Omron CX-Programmer project 新工程 (CX-Programmer 9.42)

# PLC HJ正压氦检: CJ2M CPU34
I/O table (CPU CJ2M-CPU34): rack 0 slot 0 CJ1W-NC413; rack 0 slot 1 CJ1W-SCU21-V1; rack 0 slot 2 CJ1W-AD081-V1; rack 0 slot 3 CJ1W-ID261; rack 0 slot 4 CJ1W-ID261; rack 0 slot 5 CJ1W-OD261; rack 0 slot 6 CJ1W-OD261; rack 0 slot 11 CJ2M-EIP21

## Global symbols (name address type ; comment)
0.00 BOOL  ; 扫码有料感应
0.01 BOOL  ; 抓料有料感应
0.02 BOOL  ; 下料拉带有料感应
0.03 BOOL  ; 入料托盘上料处有料
0.04 BOOL  ; 前出料托盘处有料
0.05 BOOL  ; 后出料托盘处有料
0.06 BOOL  ; 前腔体有料感应
0.07 BOOL  ; 后腔体有料感应
0.08 BOOL  ; #1腔体有料感应
0.09 BOOL  ; #2腔体有料感应
0.10 BOOL  ; 隔离处有料感应
0.11 BOOL  ; #4腔体有料感应
0.12 BOOL  ; 扫码NG#1托盘有料
0.13 BOOL  ; 扫码NG#2托盘有料
0.14 BOOL  ; 扫码NG#3托盘有料
0.15 BOOL  ; 扫码NG#4托盘有料
100.00 BOOL  ; PLC上电
100.01 BOOL  ; 紧急停止
100.02 BOOL  ; 自动启动
100.03 BOOL  ; 自动停止
100.04 BOOL  ; 报警清除
100.05 BOOL  ; 停止中
100.06 BOOL  ; 异常报警停止
100.07 BOOL  ; 关自动
100.08 BOOL  ; 空跑模式
100.09 BOOL  ; 机台内有电池
100.10 BOOL  ; 机台有错误
100.11 BOOL  ; 报警中
100.12 BOOL  ; 三色灯-绿灯
100.13 BOOL  ; 三色灯-红灯
100.14 BOOL  ; 三色灯-黄灯
100.15 BOOL  ; 三色灯-蜂鸣器
101.00 BOOL  ; 整机在初始位
101.01 BOOL  ; 电池异常中
101.03 BOOL  ; 临时暂停标志
101.04 BOOL  ; 停止互锁
101.06 BOOL  ; 腔体离线报警
10.00 BOOL  ; 下料横移气缸缩回
10.01 BOOL  ; 下料横移气缸伸出
10.02 BOOL  ; 前进料腔体托盘顶升气缸
10.03 BOOL  ; 后进料腔体托盘顶升气缸
10.04 BOOL  ; 前出料腔体托盘顶升气缸
10.05 BOOL  ; 空气净化器启动
10.06 BOOL  ; 前腔体进料夹爪气缸
10.07 BOOL  ; 前腔体进料升降气缸
10.08 BOOL  ; 后腔体进料夹爪气缸
10.09 BOOL  ; 后腔体进料升降气缸
10.10 BOOL  ; 前腔体出料夹爪气缸
10.11 BOOL  ; 前腔体出料升降气缸
10.12 BOOL  ; 后腔体出料夹爪气缸
10.13 BOOL  ; 后腔体出料升降气缸
10.14 BOOL  ; #1腔体移栽气缸伸出
10.15 BOOL  ; #1腔体移栽气缸缩回
1101.00 BOOL  ; #1腔氦检阀打开条件
1101.01 BOOL  ; #1腔氦检阀关闭条件
1101.02 BOOL  ; #1腔吹气自动启动条件
1101.03 BOOL  ; #1腔吹气自动停止条件
1102.00 BOOL  ; #2腔氦检阀打开条件
1102.01 BOOL  ; #2腔氦检阀关闭条件
1102.02 BOOL  ; #2腔吹气自动启动条件
1102.03 BOOL  ; #2腔吹气自动停止条件
1103.00 BOOL  ; #3腔氦检阀打开条件
1103.01 BOOL  ; #3腔氦检阀关闭条件
1103.02 BOOL  ; #3腔吹气自动启动条件
1103.03 BOOL  ; #3腔吹气自动停止条件
1104.00 BOOL  ; #4腔氦检阀打开条件
1104.01 BOOL  ; #4腔氦检阀关闭条件
1104.02 BOOL  ; #4腔吹气自动启动条件
1104.03 BOOL  ; #4腔吹气自动停止条件
110.01 BOOL  ; 1#腔体自检步进条件
110.15 BOOL  ; 1#腔体自检步进
111 CHANNEL  ; 1#腔体自检步序
111.00 BOOL  ; 1#腔体自检启动
111.01 BOOL  ; 真空泵打开(1#腔自检)
111.02 BOOL  ; 腔体1平移气缸后退(自检)
111.03 BOOL  ; 腔体1顶升气缸上升(自检)
111.04 BOOL  ; 腔体1抽真空(自检)
111.05 BOOL  ; 腔体1自检保压前延时
111.06 BOOL  ; 腔体1自检保压
111.07 BOOL  ; 空
111.08 BOOL  ; 1#腔体自检破真空
111.09 BOOL  ; 腔体1顶升气缸下降(自检)
111.10 BOOL  ; 腔体1平移气缸前进(自检)
111.14 BOOL  ; 1#腔体自检完成
111.15 BOOL  ; 1#腔体自检完成
112.01 BOOL  ; 2#腔体自检步进条件
112.15 BOOL  ; 2#腔体自检步进
113 CHANNEL  ; 2#腔体自检步序
113.00 BOOL  ; 2#腔体自检启动
113.01 BOOL  ; 真空泵打开(2#腔自检)
113.02 BOOL  ; 腔体2平移气缸后退(自检)
113.03 BOOL  ; 腔体2顶升气缸上升(自检)
113.04 BOOL  ; 腔体2抽真空(自检)
113.05 BOOL  ; 腔体2自检保压前延时
113.06 BOOL  ; 腔体2自检保压
113.07 BOOL  ; 空
113.08 BOOL  ; 2#腔体自检破真空
113.09 BOOL  ; 腔体2顶升气缸下降(自检)
113.10 BOOL  ; 腔体2平移气缸前进(自检)
113.14 BOOL  ; 2#腔体自检完成
113.15 BOOL  ; 2#腔体自检完成
114.01 BOOL  ; 3#腔体自检步进条件
114.15 BOOL  ; 3#腔体自检步进
115 CHANNEL  ; 3#腔体自检步序
115.00 BOOL  ; 3#腔体自检启动(自检步)
115.01 BOOL  ; 真空泵2启动
115.02 BOOL  ; 腔体3平移气缸后退(自检步)打开(3#腔自检)
115.03 BOOL  ; 腔体3顶升气缸上升
115.04 BOOL  ; 腔体3抽真空(自检步)
115.05 BOOL  ; 腔体3自检保压前延时(自检步)
115.06 BOOL  ; 腔体3自检保压(自检步)
115.07 BOOL  ; 空(自检步)
115.08 BOOL  ; 3#腔体自检破真空(自检步)
115.09 BOOL  ; 腔体3顶升气缸下降(自检步)
115.10 BOOL  ; 腔体3平移气缸前进(自检步)
115.11 BOOL  ; (自检步)
115.12 BOOL  ; (自检步)
115.13 BOOL  ; (自检步)
115.14 BOOL  ; 3#腔体自检完成(自检步)
115.15 BOOL  ; 3#腔体自检完成(自检步)
116.01 BOOL  ; 4#腔体自检步进条件
116.15 BOOL  ; 4#腔体自检步进
117 CHANNEL  ; 4#腔体自检步序
117.00 BOOL  ; 4#腔体自检启动
117.01 BOOL  ; 真空泵打开(4#腔自检)
117.02 BOOL  ; 腔体4平移气缸后退(自检)
117.03 BOOL  ; 腔体4顶升气缸上升(自检)
117.04 BOOL  ; 腔体4抽真空(自检)
117.05 BOOL  ; 腔体4自检保压前延时
117.06 BOOL  ; 腔体4自检保压
117.07 BOOL  ; 空
117.08 BOOL  ; 4#腔体自检破真空
117.09 BOOL  ; 腔体4顶升气缸下降(自检)
117.10 BOOL  ; 腔体4平移气缸前进(自检)
117.14 BOOL  ; 4#腔体自检完成
117.15 BOOL  ; 4#腔体自检完成
11.00 BOOL  ; #1腔体顶升气缸缩回
11.01 BOOL  ; #1腔体顶升气缸伸出
11.02 BOOL  ; #1腔体抽气阀
11.03 BOOL  ; #1腔体破真空阀
11.04 BOOL  ; #1腔体吹气阀
11.05 BOOL  ; #1腔体氦检阀
11.06 BOOL  ; #1电池抽气阀
11.07 BOOL  ; #1电池充氦阀
11.08 BOOL  ; #1电池破真空阀
11.09 BOOL  ; #2腔体移栽气缸缩回
11.10 BOOL  ; #2腔体移栽气缸伸出
11.11 BOOL  ; #2腔体顶升气缸缩回
11.12 BOOL  ; #2腔体顶升气缸伸出
11.13 BOOL  ; #2腔体抽气阀
11.14 BOOL  ; #2腔体破真空阀
11.15 BOOL  ; #2腔体吹气阀
120.02 BOOL  ; 清料停机条件1
120.03 BOOL  ; 清料中
121.00 BOOL  ; 整机复位(M)
121.01 BOOL  ; 进料机构复位(M)
121.02 BOOL  ; 前上料机构复位(M)
121.03 BOOL  ; 前下料机构复位(M)
121.04 BOOL  ; 后上料机构复位(M)
121.05 BOOL  ; 后下料机构复位(M)
121.06 BOOL  ; 腔体1机构复位(M)
121.07 BOOL  ; 腔体2机构复位(M)
121.08 BOOL  ; 腔体3机构复位(M)
121.09 BOOL  ; 腔体4机构复位(M)
121.10 BOOL  ; 出料机构复位(M)
1230.00 BOOL  ; 进料阻挡气缸阻挡(A)
1230.01 BOOL  ; 扫码阻挡气缸放行(A)
1230.02 BOOL  ; 扫码阻挡伸出
1230.03 BOOL  ; 扫码气缸前进(A)
1230.06 BOOL  ; 隔离气缸夹紧
1230.07 BOOL  ; 隔离气缸松开
1230.08 BOOL  ; 进料夹爪气缸张开(A)
1230.09 BOOL  ; 进料夹爪气缸夹紧(A)
1230.10 BOOL  ; 前进料旋转气缸转回(A)
1230.11 BOOL  ; 前进料旋转气缸旋转(A)
1230.12 BOOL  ; 后进料旋转气缸转回(A)
1230.13 BOOL  ; 后进料旋转气缸旋转(A)
1230.14 BOOL  ; 避位气缸接料(A)
1230.15 BOOL  ; 避位气缸避位(A)
1231.00 BOOL  ; 接料气缸前进(A)
1231.01 BOOL  ; 接料气缸后退(A)
1231.02 BOOL  ; 间隔气缸上升(A)
1231.03 BOOL  ; 间隔气缸下降(A)
1231.04 BOOL  ; 左扫码(A)
1231.05 BOOL  ; 右扫码(A)
1231.06 BOOL  ; 扫码气缸前进(A)
1231.07 BOOL  ; 扫码气缸后退(A)
1232.00 BOOL  ; 进料伺服归零(A)
1232.01 BOOL  ; 进料伺服点动前进(A)
1232.02 BOOL  ; 进料伺服点动后退(A)
1232.03 BOOL  ; 进料伺服到等待位置(A)
1232.04 BOOL  ; 进料伺服到取料位置(A)
1232.05 BOOL  ; 进料伺服到前放料位置(A)
1232.06 BOOL  ; 进料伺服到后放料位置(A)
1232.07 BOOL  ; 进料伺服到拉带安全位(A)
1232.11 BOOL  ; 进料伺服自动定位条件
1232.12 BOOL  ; 进料伺服自动定位(A)
1232.13 BOOL  ; 进料伺服自动定位
1233.00 BOOL  ; 前上料1级升降气缸上升(A)
1233.01 BOOL  ; 前上料1级升降气缸下降(A)
1233.02 BOOL  ; 前上料2级升降气缸上升(A)
1233.03 BOOL  ; 前上料2级升降气缸下降(A)
1233.04 BOOL  ; 前上料夹爪气缸夹紧(A)
1233.05 BOOL  ; 前上料夹爪气缸松开(A)
1234.00 BOOL  ; 前上料伺服归零(A)
1234.01 BOOL  ; 前上料伺服点动前进(A)
1234.02 BOOL  ; 前上料伺服点动后退(A)
1234.03 BOOL  ; 前上料伺服到等待位置(A)
1234.04 BOOL  ; 前上料伺服到取料位置(A)
1234.05 BOOL  ; 前上料伺服到仓1放料位置(A)
1234.06 BOOL  ; 前上料伺服到仓2放料位置(A)
1234.11 BOOL  ; 前上料伺服自动定位条件
1234.12 BOOL  ; 前上料伺服自动定位(A)
1235.00 BOOL  ; 前下料升降气缸上升(A)
1235.01 BOOL  ; 前下料升降气缸下降(A)
1235.02 BOOL  ; 前下料2级升降气缸上升(A)
1235.03 BOOL  ; 前下料2级升降气缸下降(A)
1235.04 BOOL  ; 前下料夹爪气缸夹紧(A)
1235.05 BOOL  ; 前下料夹爪气缸松开(A)
1236.00 BOOL  ; 前下料伺服归零(A)
1236.01 BOOL  ; 前下料伺服点动前进(A)
1236.02 BOOL  ; 前下料伺服点动后退(A)
1236.03 BOOL  ; 前下料伺服到等待位置(A)
1236.04 BOOL  ; 前下料伺服到仓1取料位置(A)
1236.05 BOOL  ; 前下料伺服到仓2取料位置(A)
1236.06 BOOL  ; 前下料伺服到放料位置(A)
1236.07 BOOL  ; 前下料伺服到NG放料位(A)
1236.09 BOOL  ; 离开#2号
1236.10 BOOL  ; 前上料伺服到仓2放料
1236.11 BOOL  ; 前下料伺服自动定位条件
1236.12 BOOL  ; 前下料伺服自动定位(A)
1237.00 BOOL  ; 后上料升降气缸上升(A)
1237.01 BOOL  ; 后上料升降气缸下降(A)
1237.02 BOOL  ; 后上料2级升降气缸上升(A)
1237.03 BOOL  ; 后上料2级升降气缸下降(A)
1237.04 BOOL  ; 后上料夹爪气缸夹紧(A)
1237.05 BOOL  ; 后上料夹爪气缸松开(A)
1238.03 BOOL  ; 后上料伺服到等待位置(A)
1238.04 BOOL  ; 后上料伺服到取料位置(A)
1238.05 BOOL  ; 后上料伺服到仓3放料位置(A)
1238.06 BOOL  ; 后上料伺服到仓4放料位置(A)
1238.09 BOOL  ; 离开#4号放料
1238.10 BOOL  ; 到#4号放料
1238.11 BOOL  ; 后上料伺服自动定位条件
1238.12 BOOL  ; 后上料伺服自动定位(A)
1239.00 BOOL  ; 后下料升降气缸上升(A)
1239.01 BOOL  ; 后下料升降气缸下降(A)
1239.02 BOOL  ; 后下料2级升降气缸上升(A)
1239.03 BOOL  ; 后下料2级升降气缸下降(A)
1239.04 BOOL  ; 后下料夹爪气缸夹紧(A)
1239.05 BOOL  ; 后下料夹爪气缸松开(A)
1240.03 BOOL  ; 后下料伺服到等待位置(A)
1240.04 BOOL  ; 后下料伺服到仓3取料位置(A)
1240.05 BOOL  ; 后下料伺服到仓4取料位置(A)
1240.06 BOOL  ; 后下料伺服到OK放料位置(A)
1240.07 BOOL  ; 后下料伺服到NG放料位置(A)
1240.11 BOOL  ; 后下料伺服自动定位条件
1240.12 BOOL  ; 后下料伺服自动定位(A)
1241.04 BOOL  ; 出料升降气缸上升(A)
1241.05 BOOL  ; 出料升降气缸下降(A)
1241.06 BOOL  ; 出料平移气缸开(A)
1241.07 BOOL  ; 出料平移气缸合(A)
1241.08 BOOL  ; 出料夹爪气缸张开(A)
1241.09 BOOL  ; 出料夹爪气缸夹紧(A)
1241.10 BOOL  ; 前出料旋转气缸初位(A)
1241.11 BOOL  ; 前出料旋转气缸旋转(A)
1241.12 BOOL  ; 后出料旋转气缸初位(A)
1241.13 BOOL  ; 后出料旋转气缸旋转(A)
1241.14 BOOL  ; 前NG气缸前进(A)
1241.15 BOOL  ; 前NG气缸后退(A)
1242.00 BOOL  ; 后NG气缸前进(A)
1242.01 BOOL  ; 后NG气缸后退(A)
1243.00 BOOL  ; 出料伺服归零(A)
1243.01 BOOL  ; 出料伺服点动前进(A)
1243.02 BOOL  ; 出料伺服点动后退(A)
1243.03 BOOL  ; 出料伺服到等待位置(A)
1243.04 BOOL  ; 出料伺服到前取料位置(A)
1243.05 BOOL  ; 出料伺服到后放料位置(A)
1243.06 BOOL  ; 出料伺服到放料位置(A)
1243.11 BOOL  ; 出料伺服自动定位条件
1243.12 BOOL  ; 出料伺服自动定位(A)
1243.13 BOOL  ; 出料伺服自动定位
1244.00 BOOL  ; 真空泵1启动(A)
1244.01 BOOL  ; 真空泵停止(A)
1244.02 BOOL  ; 吹气启动(A)
1244.03 BOOL  ; 吹气停止(A)
1244.04 BOOL  ; 氦检仪启动(A)
1244.05 BOOL  ; 氦检仪停止(A)
1244.06 BOOL  ; 真空泵2启动(A)
1245.00 BOOL  ; #1腔平移气缸前进(A)
1245.01 BOOL  ; #1腔平移气缸后退(A)
1245.02 BOOL  ; #1腔顶升气缸上升(A)
1245.03 BOOL  ; #1腔顶升气缸下降(A)
1245.04 BOOL  ; #1腔密封气缸上升(A)
1245.05 BOOL  ; #1腔密封气缸下降(A)
1245.06 BOOL  ; #1腔电池抽气阀打开(A)
1245.07 BOOL  ; #1腔电池抽气阀关闭(A)
1245.08 BOOL  ; #1腔腔体抽气阀打开(A)
1245.09 BOOL  ; #1腔腔体抽气阀关闭(A)
1245.10 BOOL  ; #1腔电池破真空阀打开(A)
1245.11 BOOL  ; #1腔电池破真空阀关闭(A)
1245.12 BOOL  ; #1腔腔体破真空阀打开(A)
1245.13 BOOL  ; #1腔腔体破真空阀关闭(A)
1245.14 BOOL  ; #1腔注氦气阀打开(A)
1245.15 BOOL  ; #1腔注氦气阀关闭(A)
1246.00 BOOL  ; #1腔氦检阀打开(A)
1246.01 BOOL  ; #1腔氦检阀关闭(A)
1246.02 BOOL  ; #1腔腔体自检启动(A)
1246.03 BOOL  ; #1腔腔体自检停止(A)
1246.04 BOOL  ; #1腔吹气启动(A)
1246.05 BOOL  ; #1腔吹气停止(A)
1247.00 BOOL  ; #2腔平移气缸前进(A)
1247.01 BOOL  ; #2腔平移气缸后退(A)
1247.02 BOOL  ; #2腔顶升气缸上升(A)
1247.03 BOOL  ; #2腔顶升气缸下降(A)
1247.04 BOOL  ; #2腔密封气缸上升(A)
1247.05 BOOL  ; #2腔密封气缸下降(A)
1247.06 BOOL  ; #2腔电池抽气阀打开(A)
1247.07 BOOL  ; #2腔电池抽气阀关闭(A)
1247.08 BOOL  ; #2腔腔体抽气阀打开(A)
1247.09 BOOL  ; #2腔腔体抽气阀关闭(A)
1247.10 BOOL  ; #2腔电池破真空阀打开(A)
1247.11 BOOL  ; #2腔电池破真空阀关闭(A)
1247.12 BOOL  ; #2腔腔体破真空阀打开(A)
1247.13 BOOL  ; #2腔腔体破真空阀关闭(A)
1247.14 BOOL  ; #2腔注氦气阀打开(A)
1247.15 BOOL  ; #2腔注氦气阀关闭(A)
1248.00 BOOL  ; #2腔氦检阀打开(A)
1248.01 BOOL  ; #2腔氦检阀关闭(A)
1248.02 BOOL  ; #2腔腔体自检启动(A)
1248.03 BOOL  ; #2腔腔体自检停止(A)
1248.04 BOOL  ; #2腔吹气启动(A)
1248.05 BOOL  ; #2腔吹气停止(A)
1249.00 BOOL  ; #3腔平移气缸前进(A)
1249.01 BOOL  ; #3腔平移气缸后退(A)
1249.02 BOOL  ; #3腔顶升气缸上升(A)
1249.03 BOOL  ; #3腔顶升气缸下降(A)
1249.04 BOOL  ; #3腔密封气缸上升(A)
1249.05 BOOL  ; #3腔密封气缸下降(A)
1249.06 BOOL  ; #3腔电池抽气阀打开(A)
1249.07 BOOL  ; #3腔电池抽气阀关闭(A)
1249.08 BOOL  ; #3腔腔体抽气阀打开(A)
1249.09 BOOL  ; #3腔腔体抽气阀关闭(A)
1249.10 BOOL  ; #3腔电池破真空阀打开(A)
1249.11 BOOL  ; #3腔电池破真空阀关闭(A)
1249.12 BOOL  ; #3腔腔体破真空阀打开(A)
1249.13 BOOL  ; #3腔腔体破真空阀关闭(A)
1249.14 BOOL  ; #3腔注氦气阀打开(A)
1249.15 BOOL  ; #3腔注氦气阀关闭(A)
1250.00 BOOL  ; #3腔氦检阀打开(A)
1250.01 BOOL  ; #3腔氦检阀关闭(A)
1250.02 BOOL  ; #3腔腔体自检启动(A)
1250.03 BOOL  ; #3腔腔体自检停止(A)
1250.04 BOOL  ; #3腔吹气启动(A)
1250.05 BOOL  ; #3腔吹气停止(A)
1251.00 BOOL  ; #4腔平移气缸前进(A)
1251.01 BOOL  ; #4腔平移气缸后退(A)
1251.02 BOOL  ; #4腔顶升气缸上升(A)
1251.03 BOOL  ; #4腔顶升气缸下降(A)
1251.04 BOOL  ; #4腔密封气缸上升(A)
1251.05 BOOL  ; #4腔密封气缸下降(A)
1251.06 BOOL  ; #4腔电池抽气阀打开(A)
1251.07 BOOL  ; #4腔电池抽气阀关闭(A)
1251.08 BOOL  ; #4腔腔体抽气阀打开(A)
1251.09 BOOL  ; #4腔腔体抽气阀关闭(A)
1251.10 BOOL  ; #4腔电池破真空阀打开(A)
1251.11 BOOL  ; #4腔电池破真空阀关闭(A)
1251.12 BOOL  ; #4腔腔体破真空阀打开(A)
1251.13 BOOL  ; #4腔腔体破真空阀关闭(A)
1251.14 BOOL  ; #4腔注氦气阀打开(A)
1251.15 BOOL  ; #4腔注氦气阀关闭(A)
1252.00 BOOL  ; #4腔氦检阀打开(A)
1252.01 BOOL  ; #4腔氦检阀关闭(A)
1252.02 BOOL  ; #4腔腔体自检启动(A)
1252.03 BOOL  ; #4腔腔体自检停止(A)
1252.04 BOOL  ; #4腔吹气启动(A)
1252.05 BOOL  ; #4腔吹气停止(A)
1255.00 BOOL  ; #1腔体移栽气缸缩回
1255.01 BOOL  ; #1腔体移栽气缸伸出
1255.02 BOOL  ; #1腔体顶升气缸伸出
1255.03 BOOL  ; #1腔体顶升气缸缩回
1257.00 BOOL  ; #2腔体移栽气缸缩回
1257.01 BOOL  ; #2腔体移栽气缸伸出
1257.02 BOOL  ; #2腔体顶升气缸伸出
1257.03 BOOL  ; #2腔体顶升气缸缩回
1259.00 BOOL  ; #3腔体移栽气缸缩回.
1259.01 BOOL  ; #3腔体移栽气缸伸出0
1259.02 BOOL  ; #3腔体顶升气缸伸出
1259.03 BOOL  ; #3腔体顶升气缸缩回
1261.00 BOOL  ; #4腔体移栽气缸缩回
1261.01 BOOL  ; #4腔体移栽气缸伸出
1261.02 BOOL  ; #4腔体顶升气缸伸出
1261.03 BOOL  ; #4腔体顶升气缸缩回
1280.00 BOOL  ; 1#腔体清氦步序自动条件
1280.01 BOOL  ; 1#腔体清氦步进条件
1280.15 BOOL  ; 1#腔体清氦步进
1281.00 BOOL  ; #1模组清氦步序开始(步)
1281.01 BOOL  ; #1模组清氦抽真空(步)
1281.02 BOOL  ; #1模组清氦抽真空阀关闭(步)
1281.03 BOOL  ; #1模组(清氦步)
1281.04 BOOL  ; #1模组计数(清氦步)
1281.05 BOOL  ; #1模组氦检阀打开(清氦步)
1281.06 BOOL  ; #1模组关氦检阀(清氦步)
1281.07 BOOL  ; #1模组破真空(清氦步)
1281.08 BOOL  ; #1模组动作选择(清氦步)
1281.09 BOOL  ; #1模组电池抽真空(清氦步)
1281.10 BOOL  ; #1模组电池抽真空阀关闭(清氦步)
1281.11 BOOL  ; #1模组电池破真空(清氦步)
1281.12 BOOL  ; #1模组清氦完成(清氦步)
1282.00 BOOL  ; #2腔体清氦步序自动条件
1282.01 BOOL  ; #2腔体清氦步进条件
1282.15 BOOL  ; #2腔体清氦步进
1283.00 BOOL  ; #2模组清氦步序开始(步)
1283.01 BOOL  ; #2模组清氦抽真空(步)
1283.02 BOOL  ; #2模组清氦抽真空阀关闭(步)
1283.03 BOOL  ; #2模组(清氦步)
1283.04 BOOL  ; #2模组计数(清氦步)
1283.05 BOOL  ; #2模组氦检阀打开(清氦步)
1283.06 BOOL  ; #2模组关氦检阀(清氦步)
1283.07 BOOL  ; #2模组破真空(清氦步)
1283.08 BOOL  ; #2模组动作选择(清氦步)
1283.09 BOOL  ; #2模组电池抽真空(清氦步)
1283.10 BOOL  ; #2模组电池抽真空阀关闭(清氦步)
1283.11 BOOL  ; #2模组电池破真空(清氦步)
1283.12 BOOL  ; #2模组清氦完成(清氦步)
1284.00 BOOL  ; #3腔体清氦步序自动条件
1284.01 BOOL  ; #3腔体清氦步进条件
1284.15 BOOL  ; #3腔体清氦步进
1285.00 BOOL  ; #3模组清氦步序开始(步)
1285.01 BOOL  ; #3模组清氦抽真空(步)
1285.02 BOOL  ; #3模组清氦抽真空阀关闭(步)
1285.03 BOOL  ; #3模组(清氦步)
1285.04 BOOL  ; #3模组计数(清氦步)
1285.05 BOOL  ; #3模组氦检阀打开(清氦步)
1285.06 BOOL  ; #3模组关氦检阀(清氦步)
1285.07 BOOL  ; #3模组破真空(清氦步)
1285.08 BOOL  ; #3模组动作选择(清氦步)
1285.09 BOOL  ; #3模组电池抽真空(清氦步)
1285.10 BOOL  ; #3模组电池抽真空阀关闭(清氦步)
1285.11 BOOL  ; #3模组电池破真空(清氦步)
1285.12 BOOL  ; #3模组清氦完成(清氦步)
1286.00 BOOL  ; #4腔体清氦步序自动条件
1286.01 BOOL  ; #4腔体清氦步进条件
1286.15 BOOL  ; #4腔体清氦步进
1287.00 BOOL  ; #4模组清氦步序开始(步)
1287.01 BOOL  ; #4模组清氦抽真空(步)
1287.02 BOOL  ; #4模组清氦抽真空阀关闭(步)
1287.03 BOOL  ; #4模组(清氦步)
1287.04 BOOL  ; #4模组计数(清氦步)
1287.05 BOOL  ; #4模组氦检阀打开(清氦步)
1287.06 BOOL  ; #4模组关氦检阀(清氦步)
1287.07 BOOL  ; #4模组破真空(清氦步)
1287.08 BOOL  ; #4模组动作选择(清氦步)
1287.09 BOOL  ; #4模组电池抽真空(清氦步)
1287.10 BOOL  ; #4模组电池抽真空阀关闭(清氦步)
1287.11 BOOL  ; #4模组电池破真空(清氦步)
1287.12 BOOL  ; #4模组清氦完成(清氦步)
12.00 BOOL  ; #2腔体氦检阀
12.01 BOOL  ; #2电池抽气阀
12.02 BOOL  ; #2电池充氦阀
12.03 BOOL  ; #2电池破真空阀
12.04 BOOL  ; #3腔体移栽气缸伸出0
12.05 BOOL  ; #3腔体移栽气缸缩回.
12.06 BOOL  ; #3腔体顶升气缸缩回
12.07 BOOL  ; #3腔体顶升气缸伸出
12.08 BOOL  ; #3腔体抽气阀
12.09 BOOL  ; #3腔体破真空阀
12.10 BOOL  ; #3腔体吹气阀
12.11 BOOL  ; #3腔体氦检阀
12.12 BOOL  ; #3电池抽气阀
12.13 BOOL  ; #3电池充氦阀
12.14 BOOL  ; #3电池破真空阀
12.15 BOOL  ; #4腔体移栽气缸伸出
130.00 BOOL  ; 进料阻挡气缸阻挡(M)
130.01 BOOL  ; 进料阻挡气缸放行(M)
130.02 BOOL  ; 扫码阻挡气缸缩回(M)
130.03 BOOL  ; 扫码阻挡气缸伸出(M)
130.04 BOOL  ; 进料升降气缸上升(M)
130.05 BOOL  ; 进料升降气缸下降(M)
130.06 BOOL  ; 进料平移气缸开(M)
130.07 BOOL  ; 进料平移气缸合(M)
130.08 BOOL  ; 进料夹爪气缸张开(M)
130.09 BOOL  ; 进料夹爪气缸夹紧(M)
130.10 BOOL  ; 下料横移气缸缩回.
130.11 BOOL  ; 下料横移气缸伸出
130.12 BOOL  ; 后进料旋转气缸转回(M)
130.13 BOOL  ; 后进料旋转气缸旋转(M)
130.14 BOOL  ; #1扫码NG气缸缩回(M)
130.15 BOOL  ; #1扫码NG气缸伸出(M)
131.00 BOOL  ; 接料气缸前进接料(M)
131.01 BOOL  ; 接料气缸后退(M)
131.02 BOOL  ; #2扫码NG气缸上升(M)
131.03 BOOL  ; #2扫码NG气缸下降(M)
131.04 BOOL  ; 左扫码(M)
131.05 BOOL  ; 右扫码(M)
131.06 BOOL  ; 扫码气缸前进(M)
131.07 BOOL  ; 扫码气缸后退(M)
131.08 BOOL  ; 夹紧阻挡气缸松开
131.09 BOOL  ; 夹紧阻挡气缸夹紧
131.10 BOOL  ; 进料#1扫码NG位置
131.11 BOOL  ; 进料#2扫码NG位置
131.12 BOOL  ; 进料#3扫码NG位置
1321.00 BOOL  ; 整机复位(Lamp)
1321.03 BOOL  ; 停止中(Lamp)
1321.05 BOOL  ; 清料停止中(Lamp)
132.00 BOOL  ; 进料伺服归零(M)
132.01 BOOL  ; 进料伺服点动前进(M)
132.02 BOOL  ; 进料伺服点动后退(M)
132.03 BOOL  ; 进料#4扫码NG位
132.04 BOOL  ; 进料伺服到取料位置(M)
132.05 BOOL  ; 进料伺服到前放料位置(M)
132.06 BOOL  ; 进料伺服到后放料位置(M)
132.07 BOOL  ; 进料伺服到拉带安全位(M)
132.09 BOOL  ; 进料升降伺服位置设定开关(M)
132.10 BOOL  ; 进料伺服位置设定开关(M)
132.11 BOOL  ; 进料伺服手动定位条件
132.12 BOOL  ; 进料伺服手动定位(M)
132.13 BOOL  ; 进料伺服手动定位
132.15 BOOL  ; 进料机构复位(M)
1330.00 BOOL  ; 进料阻挡气缸阻挡(Lamp)
1330.01 BOOL  ; 进料阻挡气缸放行(Lamp)
1330.02 BOOL  ; 扫码气缸后退(Lamp)
1330.03 BOOL  ; 扫码气缸前进(Lamp)
1330.04 BOOL  ; 进料升降气缸上升(Lamp)
1330.05 BOOL  ; 进料升降气缸下降(Lamp)
1330.06 BOOL  ; 进料平移气缸开(Lamp)
1330.07 BOOL  ; 进料平移气缸合(Lamp)
1330.08 BOOL  ; 进料夹爪气缸张开(Lamp)
1330.09 BOOL  ; 进料夹爪气缸夹紧(Lamp)
1330.10 BOOL  ; 前进料旋转气缸转回(Lamp)
1330.11 BOOL  ; 前进料旋转气缸旋转(Lamp)
1330.12 BOOL  ; 后进料旋转气缸转回(Lamp)
1330.13 BOOL  ; 后进料旋转气缸旋转(Lamp)
1330.14 BOOL  ; 避位气缸接料(Lamp)
1330.15 BOOL  ; 避位气缸伸出避位(Lamp)
1331.00 BOOL  ; 接料气缸前进(Lamp)
1331.01 BOOL  ; 接料气缸后退(Lamp)
1331.02 BOOL  ; 间隔气缸上升(Lamp)
1331.03 BOOL  ; 间隔气缸下降(Lamp)
1331.04 BOOL  ; 左扫码(Lamp)
1331.05 BOOL  ; 右扫码(Lamp)
1332.00 BOOL  ; 进料伺服归零(Lamp)
1332.01 BOOL  ; 进料伺服点动前进(Lamp)
1332.02 BOOL  ; 进料伺服点动后退(Lamp)
1332.03 BOOL  ; 进料伺服到等待位置(Lamp)
1332.04 BOOL  ; 进料伺服到取料位置(Lamp)
1332.05 BOOL  ; 进料伺服到前放料位置(Lamp)
1332.06 BOOL  ; 进料伺服到后放料位置(Lamp)
1332.07 BOOL  ; 进料伺服到拉带安全位(Lamp)
1332.09 BOOL  ; 进料伺服等待位设定(Lamp)
1332.10 BOOL  ; 进料伺服取料位设定(Lamp)
1332.11 BOOL  ; 进料伺服前放料位设定(Lamp)
1332.12 BOOL  ; 进料伺服后放料位设定(Lamp)
1332.15 BOOL  ; 进料机构复位(Lamp)
1333.00 BOOL  ; 前上料1级升降气缸下降(Lamp)
1333.01 BOOL  ; 前上料夹爪气缸夹紧(Lamp)
1333.02 BOOL  ; 前上料2级升降气缸上升(Lamp)
1333.03 BOOL  ; 前上料2级升降气缸下降(Lamp)
1333.04 BOOL  ; 前上料夹爪气缸夹紧(Lamp)
1333.05 BOOL  ; 前上料夹爪气缸松开(Lamp)
1334.00 BOOL  ; 前上料伺服归零(Lamp)
1334.01 BOOL  ; 前上料伺服点动前进(Lamp)
1334.02 BOOL  ; 前上料伺服点动后退(Lamp)
1334.03 BOOL  ; 前上料伺服到等待位置(Lamp)
1334.04 BOOL  ; 前上料伺服到取料位置(Lamp)
1334.05 BOOL  ; 前上料伺服到仓1放料位置(Lamp)
1334.06 BOOL  ; 前上料伺服到仓2放料位置(Lamp)
1334.09 BOOL  ; 前上料伺服等待位设定(Lamp)
1334.10 BOOL  ; 前上料伺服取料位设定(Lamp)
1334.11 BOOL  ; 前上料伺服仓1放料位设定(Lamp)
1334.12 BOOL  ; 前上料伺服仓2放料位设定(Lamp)
1334.15 BOOL  ; 前上料机构复位(Lamp)
1335.00 BOOL  ; 前下料1级升降气缸上升(Lamp)
1335.01 BOOL  ; 前下料升降气缸下降(Lamp)
1335.02 BOOL  ; 前下料夹爪气缸夹紧(Lamp)
1335.03 BOOL  ; 前下料2级升降气缸下降(Lamp)
1335.04 BOOL  ; 前下料夹爪气缸夹紧(Lamp)
1335.05 BOOL  ; 前下料夹爪气缸松开(Lamp)
1336.00 BOOL  ; 前下料伺服归零(Lamp)
1336.01 BOOL  ; 前下料伺服点动前进(Lamp)
1336.02 BOOL  ; 前下料伺服点动后退(Lamp)
1336.03 BOOL  ; 前下料伺服到等待位置(Lamp)
1336.04 BOOL  ; 前下料伺服到仓1取料位置(Lamp)
1336.05 BOOL  ; 前下料伺服到仓2取料位置(Lamp)
1336.06 BOOL  ; 前下料伺服OK放料位置(Lamp)
1336.07 BOOL  ; 前下料伺服NG放料位置(Lamp)
1336.10 BOOL  ; 前下料伺服仓1取料位设定(Lamp)
1336.11 BOOL  ; 前下料伺服仓2取料位设定(Lamp)
1336.12 BOOL  ; 前下料伺服放料位设定(Lamp)
1336.15 BOOL  ; 前下料机构复位(Lamp)
1337.00 BOOL  ; 后上料升降气缸下降(Lamp)
1337.01 BOOL  ; 后上料夹爪气缸夹紧(Lamp)
1337.02 BOOL  ; 后上料2级升降气缸上升(Lamp)
1337.03 BOOL  ; 后上料2级升降气缸下降(Lamp)
1337.04 BOOL  ; 后上料夹爪气缸夹紧(Lamp)
1337.05 BOOL  ; 后上料夹爪气缸松开(Lamp)
1338.00 BOOL  ; 后上料伺服归零(Lamp)
1338.01 BOOL  ; 后上料伺服点动后进(Lamp)
1338.02 BOOL  ; 后上料伺服点动后退(Lamp)
1338.03 BOOL  ; 后上料伺服到等待位置(Lamp)
1338.04 BOOL  ; 后上料伺服到取料位置(Lamp)
1338.05 BOOL  ; 后上料伺服到仓1放料位置(Lamp)
1338.06 BOOL  ; 后上料伺服到仓2放料位置(Lamp)
1338.09 BOOL  ; 后上料伺服等待位设定(Lamp)
1338.10 BOOL  ; 后上料伺服取料位设定(Lamp)
1338.11 BOOL  ; 后上料伺服仓1放料位设定(Lamp)
1338.12 BOOL  ; 后上料伺服仓2放料位设定(Lamp)
1338.15 BOOL  ; 后上料机构复位(Lamp)
1339.00 BOOL  ; 后下料1级升降气缸上升(Lamp)
1339.01 BOOL  ; 后下料升降气缸下降(Lamp)
1339.02 BOOL  ; 后下料夹爪气缸夹紧(Lamp)
1339.03 BOOL  ; 后下料2级升降气缸下降(Lamp)
1339.04 BOOL  ; 后下料夹爪气缸夹紧(Lamp)
1339.05 BOOL  ; 后下料夹爪气缸松开(Lamp)
133.00 BOOL  ; 前上料升降气缸上升(M)
133.01 BOOL  ; 前上料升降气缸下降(M)
133.02 BOOL  ; 前上料2级升降气缸上升(M)
133.03 BOOL  ; 前上料2级升降气缸下降(M)
133.04 BOOL  ; 前上料夹爪气缸夹紧(M)
133.05 BOOL  ; 前上料夹爪气缸松开(M)
133.08 BOOL  ; 前上料夹爪气缸夹紧(复位)(M)
133.09 BOOL  ; 前上料夹爪气缸松开(复位)(M)
133.10 BOOL  ; 前上料升降气缸上升(复位)(M)
133.11 BOOL  ; 前上料2级升降气缸上升(复位)(M)
133.12 BOOL  ; 前上料伺服归零(复位)(M)
133.13 BOOL  ; 前上料伺服到取料位置(复位)(M)
1340.00 BOOL  ; 后下料伺服归零(Lamp)
1340.01 BOOL  ; 后下料伺服点动前进(Lamp)
1340.02 BOOL  ; 后下料伺服点动后退(Lamp)
1340.03 BOOL  ; 后下料伺服到等待位置(Lamp)
1340.04 BOOL  ; 后下料伺服到仓3取料位置(Lamp)
1340.05 BOOL  ; 后下料伺服到仓2取料位置(Lamp)
1340.06 BOOL  ; 后下料伺服到OK放料位置(Lamp)
1340.07 BOOL  ; 后下料伺服到NG放料位置(Lamp)
1340.09 BOOL  ; 后下料伺服等待位设定(Lamp)
1340.10 BOOL  ; 后下料伺服仓1取料位设定(Lamp)
1340.11 BOOL  ; 后下料伺服仓2取料位设定(Lamp)
1340.12 BOOL  ; 后下料伺服放料位设定(Lamp)
1340.15 BOOL  ; 后下料机构复位(Lamp)
1341.04 BOOL  ; 出料升降气缸上升(Lamp)
1341.05 BOOL  ; 出料升降气缸下降(Lamp)
1341.06 BOOL  ; 出料平移气缸开(Lamp)
1341.07 BOOL  ; 出料平移气缸合(Lamp)
1341.08 BOOL  ; 出料夹爪气缸张开(Lamp)
1341.09 BOOL  ; 出料夹爪气缸夹紧(Lamp)
1341.10 BOOL  ; 前出料旋转气缸初位(Lamp)
1341.11 BOOL  ; 前出料旋转气缸旋转(Lamp)
1341.12 BOOL  ; 后出料旋转气缸初位(Lamp)
1341.13 BOOL  ; 后出料旋转气缸旋转(Lamp)
1341.14 BOOL  ; 前NG气缸前进(Lamp)
1341.15 BOOL  ; 前NG气缸后退(Lamp)
1342.00 BOOL  ; 后NG气缸前进(Lamp)
1342.01 BOOL  ; 后NG气缸后退(Lamp)
1343.00 BOOL  ; 出料伺服归零(Lamp)
1343.01 BOOL  ; 出料伺服点动前进(Lamp)
1343.02 BOOL  ; 出料伺服点动后退(Lamp)
1343.03 BOOL  ; 出料伺服到等待位置(Lamp)
1343.04 BOOL  ; 出料伺服到前取料位置(Lamp)
1343.05 BOOL  ; 出料伺服到后放料位置(Lamp)
1343.06 BOOL  ; 出料伺服到放料位置(Lamp)
1343.09 BOOL  ; 出料伺服等待位设定(Lamp)
1343.10 BOOL  ; 出料伺服前取料位设定(Lamp)
1343.11 BOOL  ; 出料伺服后取料位设定(Lamp)
1343.12 BOOL  ; 出料伺服放料位设定(Lamp)
1343.15 BOOL  ; 出料机构复位(Lamp)
1344.00 BOOL  ; 真空泵启动(Lamp)
1344.01 BOOL  ; 真空泵停止(Lamp)
1344.02 BOOL  ; #1腔吹气启动(Lamp)
1344.03 BOOL  ; 吹气停止(Lamp)
1344.04 BOOL  ; 氦检仪启动(Lamp)
1344.05 BOOL  ; 氦检仪停止(Lamp)
1344.06 BOOL  ; #2吹气启动(M)
1344.07 BOOL  ; 真空泵2停止(Lamp)
1344.08 BOOL  ; #3腔体吹气阀
1345.00 BOOL  ; 自检条件不满足
1345.01 BOOL  ; #1腔平移气缸后退(Lamp)
1345.02 BOOL  ; #1腔顶升气缸上升(Lamp)
1345.03 BOOL  ; #1腔顶升气缸下降(Lamp)
1345.04 BOOL  ; #1腔密封气缸上升(Lamp)
1345.05 BOOL  ; #1腔密封气缸下降(Lamp)
1345.06 BOOL  ; #1腔电池抽气阀打开(Lamp)
1345.07 BOOL  ; #1腔电池抽气阀关闭(Lamp)
1345.08 BOOL  ; #1腔腔体抽气阀打开(Lamp)
1345.09 BOOL  ; #1腔腔体抽气阀关闭(Lamp)
1345.10 BOOL  ; #1腔电池破真空阀打开(Lamp)
1345.11 BOOL  ; #1腔电池破真空阀关闭(Lamp)
1345.12 BOOL  ; #1腔腔体破真空阀打开(Lamp)
1345.13 BOOL  ; #1腔腔体破真空阀关闭(Lamp)
1345.14 BOOL  ; #1腔注氦气阀打开(Lamp)
1345.15 BOOL  ; #1腔注氦气阀关闭(Lamp)
1346.00 BOOL  ; #1腔氦检阀打开(Lamp)
1346.01 BOOL  ; #1腔氦检阀关闭(Lamp)
1346.02 BOOL  ; #1腔腔体自检启动(Lamp)
1346.03 BOOL  ; #1腔腔体自检停止(Lamp)
1346.15 BOOL  ; #1腔机构复位(Lamp)
1347.00 BOOL  ; #2腔平移气缸后退(Lamp)
1347.01 BOOL  ; #2腔平移气缸前进(Lamp)
1347.02 BOOL  ; #2腔顶升气缸上升(Lamp)
1347.03 BOOL  ; #2腔顶升气缸下降(Lamp)
1347.04 BOOL  ; #2腔密封气缸上升(Lamp)
1347.05 BOOL  ; #2腔密封气缸下降(Lamp)
1347.06 BOOL  ; #2腔电池抽气阀打开(Lamp)
1347.07 BOOL  ; #2腔电池抽气阀关闭(Lamp)
1347.08 BOOL  ; #2腔腔体抽气阀打开(Lamp)
1347.09 BOOL  ; #2腔腔体抽气阀关闭(Lamp)
1347.10 BOOL  ; #2腔电池破真空阀打开(Lamp)
1347.11 BOOL  ; #2腔电池破真空阀关闭(Lamp)
1347.12 BOOL  ; #2腔腔体破真空阀打开(Lamp)
1347.13 BOOL  ; #2腔腔体破真空阀关闭(Lamp)
1347.14 BOOL  ; #2腔注氦气阀打开(Lamp)
1347.15 BOOL  ; #2腔注氦气阀关闭(Lamp)
1348.00 BOOL  ; #2腔氦检阀打开(Lamp)
1348.01 BOOL  ; #2腔氦检阀关闭(Lamp)
1348.02 BOOL  ; #2腔腔体自检启动(Lamp)
1348.03 BOOL  ; #2腔腔体自检停止(Lamp)
1348.15 BOOL  ; #2腔机构复位(Lamp)
1349.00 BOOL  ; #3腔平移气缸后退(Lamp)
1349.01 BOOL  ; #3腔平移气缸前进(Lamp)
1349.02 BOOL  ; #3腔顶升气缸上升(Lamp)
1349.03 BOOL  ; #3腔顶升气缸下降(Lamp)
1349.04 BOOL  ; #3腔密封气缸上升(Lamp)
1349.05 BOOL  ; #3腔密封气缸下降(Lamp)
1349.06 BOOL  ; #3腔电池抽气阀打开(Lamp)
1349.07 BOOL  ; #3腔电池抽气阀关闭(Lamp)
1349.08 BOOL  ; #3腔腔体抽气阀打开(Lamp)
1349.09 BOOL  ; #3腔腔体抽气阀关闭(Lamp)
1349.10 BOOL  ; #3腔电池破真空阀打开(Lamp)
1349.11 BOOL  ; #3腔电池破真空阀关闭(Lamp)
1349.12 BOOL  ; #3腔腔体破真空阀打开(Lamp)
1349.13 BOOL  ; #3腔腔体破真空阀关闭(Lamp)
1349.14 BOOL  ; #3腔注氦气阀打开(Lamp)
1349.15 BOOL  ; #3腔注氦气阀关闭(Lamp)
134.00 BOOL  ; 前上料伺服归零(M)
134.01 BOOL  ; 前上料伺服点动前进(M)
134.02 BOOL  ; 前上料伺服点动后退(M)
134.03 BOOL  ; 前上料伺服到等待位置(M)
134.04 BOOL  ; 前上料伺服到取料位置(M)
134.05 BOOL  ; 前上料伺服到仓1放料位置(M)
134.06 BOOL  ; 前上料伺服到仓2放料位置(M)
134.07 BOOL  ; 前上料伺服手动定位条件
134.10 BOOL  ; 前上料伺服设定打开(M)
134.11 BOOL  ; 前上料伺服手动定位条件
134.12 BOOL  ; 前上料伺服手动定位(M)
134.13 BOOL  ; 前上料伺服手动定位
134.15 BOOL  ; 前上料机构复位(M)
1350.00 BOOL  ; #3腔氦检阀打开(Lamp)
1350.01 BOOL  ; #3腔氦检阀关闭(Lamp)
1350.02 BOOL  ; #3腔腔体自检启动(Lamp)
1350.03 BOOL  ; #3腔腔体自检停止(Lamp)
1350.15 BOOL  ; #3腔机构复位(Lamp)
1351.00 BOOL  ; #4腔平移气缸后退(Lamp)
1351.01 BOOL  ; #4腔平移气缸前进(Lamp)
1351.02 BOOL  ; #4腔顶升气缸上升(Lamp)
1351.03 BOOL  ; #4腔顶升气缸下降(Lamp)
1351.04 BOOL  ; #4腔密封气缸上升(Lamp)
1351.05 BOOL  ; #4腔密封气缸下降(Lamp)
1351.06 BOOL  ; #4腔电池抽气阀打开(Lamp)
1351.07 BOOL  ; #4腔电池抽气阀关闭(Lamp)
1351.08 BOOL  ; #4腔腔体抽气阀打开(Lamp)
1351.09 BOOL  ; #4腔腔体抽气阀关闭(Lamp)
1351.10 BOOL  ; #4腔电池破真空阀打开(Lamp)
1351.11 BOOL  ; #4腔电池破真空阀关闭(Lamp)
1351.12 BOOL  ; #4腔腔体破真空阀打开(Lamp)
1351.13 BOOL  ; #4腔腔体破真空阀关闭(Lamp)
1351.14 BOOL  ; #4腔注氦气阀打开(Lamp)
1351.15 BOOL  ; #4腔注氦气阀关闭(Lamp)
1352.00 BOOL  ; #4腔氦检阀打开(Lamp)
1352.01 BOOL  ; #4腔氦检阀关闭(Lamp)
1352.02 BOOL  ; #4腔腔体自检启动(Lamp)
1352.03 BOOL  ; #4腔腔体自检停止(Lamp)
1352.15 BOOL  ; #4腔机构复位(Lamp)
135.00 BOOL  ; 前下料1级升降气缸上升(M)
135.01 BOOL  ; 前下料升降气缸下降(M)
135.02 BOOL  ; 前下料2级升降气缸上升(M)
135.03 BOOL  ; 前下料2级升降气缸下降(M)
135.04 BOOL  ; 前下料夹爪气缸夹紧(M)
135.05 BOOL  ; 前下料夹爪气缸松开(M)
135.08 BOOL  ; 前下料夹爪气缸夹紧(复位)(M)
135.09 BOOL  ; 前下料夹爪气缸松开(复位)(M)
135.10 BOOL  ; 前下料升降气缸上升(复位)(M)
135.11 BOOL  ; 前下料2级升降气缸上升(复位)(M)
135.12 BOOL  ; 前下料伺服归零(复位)(M)
135.13 BOOL  ; 前下料伺服到放料位置(复位)(M)
136.00 BOOL  ; 前下料伺服归零(M)
136.01 BOOL  ; 前下料伺服点动前进(M)
136.02 BOOL  ; 前下料伺服点动后退(M)
136.03 BOOL  ; 前下料伺服到等待位置(M)
136.04 BOOL  ; 前下料伺服到仓1取料位置(M)
136.05 BOOL  ; 前下料伺服到仓2取料位置(M)
136.06 BOOL  ; 前下料伺服到OK放料位置(M)
136.07 BOOL  ; 前下料伺服到NG放料位置(M)
136.10 BOOL  ; 前下料伺服位置设定开(M)
136.11 BOOL  ; 前下料伺服手动定位条件
136.12 BOOL  ; 前下料伺服手动定位(M)
136.13 BOOL  ; 前下料伺服手动定位
136.15 BOOL  ; 前下料机构复位(M)
1370.00 BOOL  ; 间隔气缸上升条件
1370.01 BOOL  ; 间隔气缸下降条件
1370.02 BOOL  ; 接料气缸前进条件(A)
1370.03 BOOL  ; 接料气缸后退条件(A)
1370.04 BOOL  ; 扫码气缸前进条件(A)
1370.05 BOOL  ; 扫码气缸后退条件(A)
137.00 BOOL  ; 后上料升降气缸上升(M)
137.01 BOOL  ; 后上料升降气缸下降(M)
137.02 BOOL  ; 后上料2级升降气缸上升(M)
137.03 BOOL  ; 后上料2级升降气缸下降(M)
137.04 BOOL  ; 后上料夹爪气缸夹紧(M)
137.05 BOOL  ; 后上料夹爪气缸松开(M)
137.08 BOOL  ; 后上料夹爪气缸夹紧(复位)(M)
137.09 BOOL  ; 后上料夹爪气缸松开(复位)(M)
137.10 BOOL  ; 后上料升降气缸上升(复位)(M)
137.11 BOOL  ; 后上料2级升降气缸上升(复位)(M)
137.12 BOOL  ; 后上料伺服归零(复位)(M)
137.13 BOOL  ; 后上料伺服到取料位置(复位)(M)
1380.02 BOOL  ; 进料升降伺服在取料位
1380.03 BOOL  ; 进料升降伺服在放料高度
138.00 BOOL  ; 后上料伺服归零(M)
138.01 BOOL  ; 后上料伺服点动后进(M)
138.02 BOOL  ; 后上料伺服点动后退(M)
138.03 BOOL  ; 后上料伺服到等待位置(M)
138.04 BOOL  ; 后上料伺服到取料位置(M)
138.05 BOOL  ; 后上料伺服到仓3放料位置(M)
138.06 BOOL  ; 后上料伺服到仓4放料位置(M)
138.10 BOOL  ; 后上料伺服位置设定开关(M)
138.11 BOOL  ; 后上料伺服手动定位条件
138.12 BOOL  ; 后上料伺服手动定位(M)
138.13 BOOL  ; 后上料伺服手动定位
138.15 BOOL  ; 后上料机构复位(M)
1395.02 BOOL  ; 扫码机构自动/单次条件
1396.00 BOOL  ; 自动扫码条件
1396.01 BOOL  ; 扫码步进条件
1396.15 BOOL  ; 扫码步进
1397 CHANNEL  ; 自动扫码步
1397.00 BOOL  ; 自动扫码开始
1397.01 BOOL  ; 扫码步
1397.02 BOOL  ; 扫码等待结果
1397.03 BOOL  ; MES进站
1397.04 BOOL  ; 记忆
1397.05 BOOL  ; 扫码阻挡缩回
1397.06 BOOL  ; 扫码阻挡伸出
1397.07 BOOL  ; 空
1397.08 BOOL  ; 扫码步完成
1397.09 BOOL  ; 空
1399.01 BOOL  ; 扫码条件
1399.02 BOOL  ; 扫码阻挡气缸缩回条件
1399.03 BOOL  ; 扫码阻挡气缸伸出条件
1399.06 BOOL  ; 隔离气缸夹紧条件
1399.07 BOOL  ; 隔离气缸缩回的条件
139.00 BOOL  ; 后下料升降气缸上升(M)
139.01 BOOL  ; 后下料升降气缸下降(M)
139.02 BOOL  ; 后下料2级升降气缸上升(M)
139.03 BOOL  ; 后下料2级升降气缸下降(M)
139.04 BOOL  ; 后下料夹爪气缸夹紧(M)
139.05 BOOL  ; 后下料夹爪气缸松开(M)
139.08 BOOL  ; 后下料夹爪气缸夹紧(复位)(M)
139.09 BOOL  ; 后下料夹爪气缸松开(复位)(M)
139.10 BOOL  ; 后出料机械手升降气缸上升(复位)(M)
139.11 BOOL  ; 后下料2级升降气缸上升(复位)(M)
139.12 BOOL  ; 后下料伺服归零(复位)(M)
139.13 BOOL  ; 后下料伺服到放料位置(复位)(M)
13.00 BOOL  ; #4腔体移栽气缸缩回
13.01 BOOL  ; #4腔体顶升气缸缩回
13.02 BOOL  ; #4腔体顶升气缸伸出
13.03 BOOL  ; #4腔体抽气阀
13.04 BOOL  ; #4腔体破真空阀
13.05 BOOL  ; #4腔体吹气阀
13.06 BOOL  ; #4腔体氦检阀
13.07 BOOL  ; #4电池抽气阀
13.08 BOOL  ; #4电池充氦阀
13.09 BOOL  ; #4电池破真空阀
13.10 BOOL  ; #1扫码NG推料气缸
13.11 BOOL  ; #2扫码NG推料气缸
13.12 BOOL  ; #1测试NG推料气缸
13.13 BOOL  ; #2测试NG推料气缸
13.14 BOOL  ; 进料拉带电机
13.15 BOOL  ; 出料拉带电机
1400.00 BOOL  ; 进料机构在初始位
1400.01 BOOL  ; 进料水平伺服在#4扫码NG位
1400.02 BOOL  ; 进料水平伺服在取料位置
1400.03 BOOL  ; 进料水平伺服前放料位置
1400.04 BOOL  ; 进料水平伺服在后放料位
1400.05 BOOL  ; 进料水平伺服在#1扫码NG位
1400.06 BOOL  ; 进料水平伺服在#2扫码NG位
1400.07 BOOL  ; 扫码NG缓存机构在初始位
1400.08 BOOL  ; 扫码机构在初始位
1400.09 BOOL  ; 进料机构正常停止条件
1400.10 BOOL  ; 进料机构清料停止条件
1400.11 BOOL  ; 进料水平伺服在#3扫码NG位
1400.12 BOOL  ; 到后放料位放料
1400.13 BOOL  ; 可到前上料
1400.14 BOOL  ; 到后放料条件
1400.15 BOOL  ; 进料伺服在设定位置
1401.00 BOOL  ; 进料机构有错误
1401.01 BOOL  ; 进料伺服手动定位目标位置设定OK
1401.02 BOOL  ; 进料伺服自动定位目标位置设定OK
1401.03 BOOL  ; 进料伺服到取料位条件
1401.04 BOOL  ; 进料伺服到取料位条件
1401.05 BOOL  ; 进料伺服到前放料位条件
1401.06 BOOL  ; 进料伺服到后放料位条件
1401.07 BOOL  ; 进料伺服可放料安全条件
1401.08 BOOL  ; 间隔气缸下降条件
1401.09 BOOL  ; 进料状态
1401.10 BOOL  ; 前、后上下料机械手条件
1401.11 BOOL  ; 出料状态
1401.12 BOOL  ; 前、后出料机械手状态
1401.13 BOOL  ; 到前取料条件
1401.15 BOOL  ; 到后取料条件
1402.09 BOOL  ; 进料伺服手动运转条件
1403 CHANNEL  ; 扫码自动步序
1403.00 BOOL  ; 扫码机构自动开始(步)
1403.01 BOOL  ; 扫码气缸前进(步)
1403.02 BOOL  ; 扫码(步)
1403.03 BOOL  ; 等待扫码结果(步)
1403.04 BOOL  ; 扫码气缸后退(步)
1403.05 BOOL  ; MES进站校验(步)
1403.06 BOOL  ; 扫码完成(步)
1403.07 BOOL  ; 扫码步序完成(步)
1404 CHANNEL  ; 扫码NG缓存步序
1404.00 BOOL  ; 扫码NG缓存机构自动开始(步)
1404.01 BOOL  ; 避位气缸缩回接料(步)
1404.02 BOOL  ; 接料气缸前进接料(步)
1404.03 BOOL  ; 等待进料机械手放料(步)
1404.04 BOOL  ; 避位气缸避位(步)
1404.05 BOOL  ; 间隔气缸下降隔料(步)
1404.06 BOOL  ; 接料气缸后退(步)
1404.08 BOOL  ; 间隔气缸上升复位(步)
1404.09 BOOL  ; 扫码NG缓存自动完成(步)
1405.00 BOOL  ; 进料机构单次循环
1405.01 BOOL  ; 进料机构单次循环完成
1405.02 BOOL  ; 进料机构自动/单次循环
1405.03 BOOL  ; 扫码机构单次循环完成
1405.05 BOOL  ; 扫码机构步进条件
1405.08 BOOL  ; 扫码机构自动
1405.09 BOOL  ; 扫码机构步进
1405.10 BOOL  ; 扫码NG缓存机构自动
1405.11 BOOL  ; 扫码NG缓存机构自动条件
1405.12 BOOL  ; 扫码NG缓存机构步进条件
1405.15 BOOL  ; 扫码NG缓存机构步进
1406.00 BOOL  ; 进料机构自动条件
1406.01 BOOL  ; 进料机构步进条件
1406.15 BOOL  ; 进料机构步进
1407 CHANNEL  ; 进料自动步序
1407.00 BOOL  ; 进料机构自动开始(步)
1407.01 BOOL  ; 到前|后上料位|扫码NG(步)
1407.02 BOOL  ; 等待夹紧(步)
1407.03 BOOL  ; 等待进料上升(步)
1407.04 BOOL  ; 进料伺服回上料位料(步)
1407.05 BOOL  ; 进料伺服归零(步)
1407.06 BOOL  ; 进料升降上升(步)
1407.07 BOOL  ; 进料伺服取料后到待机位(步)
1407.08 BOOL  ; 进料伺服到放料位&进料平移关闭(步)
1407.09 BOOL  ; 进料升降下降放料(步)
1407.10 BOOL  ; 进料夹爪松开(步)
1407.11 BOOL  ; 进料升降上升(步)
1407.12 BOOL  ; 进料伺服归零(步)
1407.13 BOOL  ; 进料伺服放料后到待机位(步)
1407.14 BOOL  ; 进料旋转气缸旋转(步)
1407.15 BOOL  ; 进料自动完成
1409.02 BOOL  ; 扫码阻挡气缸阻挡条件(A)
1409.03 BOOL  ; 扫码阻挡气缸放行条件(A)
1409.14 BOOL  ; 避位气缸接料条件(A)
1409.15 BOOL  ; 避位气缸避位条件(A)
140.00 BOOL  ; 后下料伺服归零(M)
140.01 BOOL  ; 后下料伺服点动前进(M)
140.02 BOOL  ; 后下料伺服点动后退(M)
140.03 BOOL  ; 后下料伺服到等待位置(M)
140.04 BOOL  ; 后下料伺服到仓3取料位置(M)
140.05 BOOL  ; 后下料伺服到仓4取料位置(M)
140.06 BOOL  ; 后下料伺服到放料位置(M)
140.07 BOOL  ; 后下料伺服到NG放料位置(M)
140.10 BOOL  ; 后下料伺位置设定开关(M)
140.11 BOOL  ; 后下料伺服手动定位条件
140.12 BOOL  ; 后下料伺服手动定位(M)
140.13 BOOL  ; 后下料伺服手动定位
140.15 BOOL  ; 后下料机构复位(M)
1410.00 BOOL  ; 前上料机构在初始位
1410.01 BOOL  ; 前上料伺服在待机位置
1410.02 BOOL  ; 前上料伺服在取料位置
1410.03 BOOL  ; 前上料伺服在仓1放料位置
1410.04 BOOL  ; 前上料伺服在仓2放料位置
1410.05 BOOL  ; 前上料伺服在原点位置
1410.06 BOOL  ; 前上料伺服在原点位置
1410.09 BOOL  ; 前上料机构正常停止条件
1410.10 BOOL  ; 前上料机构清料停止条件
1410.15 BOOL  ; 前上料伺服在设定位置
1411.00 BOOL  ; 前上料机构有错误
1411.01 BOOL  ; 前上料伺服手动定位目标位置设定OK
1411.02 BOOL  ; 前上料伺服自动定位目标位置设定OK
1411.03 BOOL  ; 前上料伺服到待机位安全条件
1411.04 BOOL  ; 前上料伺服到取料位安全条件
1411.05 BOOL  ; 前上料伺服到1#仓放料位安全条件
1411.06 BOOL  ; 前上料伺服到2#仓放料位安全条件
1411.07 BOOL  ; 上料可向腔1
1411.08 BOOL  ; 上料可向腔2
1415.00 BOOL  ; 前上料机构单次循环
1415.01 BOOL  ; 前上料机构单次循环完成
1415.02 BOOL  ; 前上料机构自动/单次循环
1416.00 BOOL  ; 前上料机构自动条件
1416.01 BOOL  ; 前上料机构步进条件
1416.15 BOOL  ; 前上料机构步进
1417 CHANNEL  ; 前上料自动步序
1417.00 BOOL  ; 前上料机构自动开始(步)
1417.01 BOOL  ; 前上料伺服到取料位(步)
1417.02 BOOL  ; 前上料升降气缸下降取料(步)
1417.03 BOOL  ; 前上料夹爪夹紧(步)
1417.04 BOOL  ; 前上料升降气缸取料后上升(步)
1417.05 BOOL  ; 前上料伺服到放料位(步)
1417.06 BOOL  ; 前上料升降气缸下降放料(步)
1417.09 BOOL  ; 前上料夹爪松开(步)
1417.10 BOOL  ; 前上料升降气缸上升(步)
1417.11 BOOL  ; 前上料伺服到取料位(步)
1417.15 BOOL  ; 前上料自动运行结束(步)
1419.00 BOOL  ; 前上料1级升降气缸上升条件
1419.02 BOOL  ; 前上料2级升降气缸上条件
141.04 BOOL  ; 出料#1升降气缸上升(M)
141.05 BOOL  ; 出料#1升降气缸下降(M)
141.06 BOOL  ; 下料横移气缸开(M)
141.07 BOOL  ; 下料横移气缸合(M)
141.08 BOOL  ; 出料夹爪气缸张开(M)
141.09 BOOL  ; 出料夹爪气缸夹紧(M)
141.10 BOOL  ; #1测试NG气缸缩回(M)
141.11 BOOL  ; #1测试NG气缸伸出(M)
141.12 BOOL  ; #2测试NG气缸缩回(M)
141.13 BOOL  ; #2测试NG气缸伸出(M)
141.14 BOOL  ; 前腔体出料顶升气缸伸出(M)
141.15 BOOL  ; 前腔体出料顶升气缸缩回(M)
1420.00 BOOL  ; 前下料机构在初始位
1420.01 BOOL  ; 前下料伺服在待机位置
1420.02 BOOL  ; 前下料伺服在仓1取料位置
1420.03 BOOL  ; 前下料伺服在仓2取料位置
1420.04 BOOL  ; 前下料伺服在放料位置
1420.05 BOOL  ; 前下料伺服在NG放料位置
1420.06 BOOL  ; 前下料伺服在原点位置
1420.09 BOOL  ; 前下料机构正常停止条件
1420.10 BOOL  ; 前下料机构清料停止条件
1420.15 BOOL  ; 前下料机构在设定位置
1421.00 BOOL  ; 前下料机构有错误
1421.01 BOOL  ; 前下料伺服手动定位目标位置设定OK
1421.02 BOOL  ; 前下料伺服自动定位目标位置设定OK
1421.03 BOOL  ; 前下料伺服到待机位条件
1421.04 BOOL  ; 前下料伺服到1#仓取料位条件
1421.05 BOOL  ; 前下料伺服到2#仓取料安全条件
1421.06 BOOL  ; 前下料伺服到放料位条件
1421.07 BOOL  ; 前下料可向腔1
1421.08 BOOL  ; 前下料可向腔2
1421.10 BOOL  ; 前下料升降气缸在放料位下降放料条件
1425.00 BOOL  ; 前下料机构单次循环
1425.01 BOOL  ; 前下料机构单次循环完成
1425.02 BOOL  ; 前下料机构自动/单次循环
1426.00 BOOL  ; 前下料机构自动条件
1426.01 BOOL  ; 前下料机构步进条件
1426.15 BOOL  ; 前下料机构步进
1427 CHANNEL  ; 前下料自动步序
1427.00 BOOL  ; 前下料机构自动开始(步)
1427.01 BOOL  ; 前下料到取料位(步)
1427.02 BOOL  ; 前下料升降下降取料(步)
1427.03 BOOL  ; 前下料夹爪夹紧(步)
1427.05 BOOL  ; 前下料升降取料后上升(步)
1427.06 BOOL  ; 前下料伺服到放料位&前出料旋转(步)
1427.07 BOOL  ; 前下料升降气缸下降放料(步)
1427.08 BOOL  ; (前下料步)
1427.09 BOOL  ; 前下料夹爪松开(步)
1427.10 BOOL  ; 前下料升降气缸放料后上升(步)
1427.11 BOOL  ; 空(步)
1427.12 BOOL  ; 空(步)
1427.13 BOOL  ; 空(步)
1427.14 BOOL  ; 前下料自动完成(步)
1429.01 BOOL  ; 前下料升降气缸下降放料条件(A)
142.00 BOOL  ; 后腔体出料顶升气缸伸出(M)
142.01 BOOL  ; 后腔体出料顶升气缸缩回(M)
142.05 BOOL  ; 前出料旋转气缸初位(复位)(M)
142.06 BOOL  ; 后出料旋转气缸初位(复位)(M)
142.07 BOOL  ; 前NG气缸前进(复位)(M)
142.08 BOOL  ; 后NG气缸前进(复位)(M)
142.09 BOOL  ; 出料升降伺位设置开关
142.10 BOOL  ; 出料水平移载伺位置设置开关
142.11 BOOL  ; 出料伺服归零(复位)(M)
142.12 BOOL  ; 出料伺服到等待位置(复位)(M)
1430.00 BOOL  ; 后上料机构在初始位
1430.01 BOOL  ; 后上料伺服在待机位置
1430.02 BOOL  ; 后上料伺服在取料位置
1430.03 BOOL  ; 后上料伺服在仓3放料位置
1430.04 BOOL  ; 后上料伺服在仓4放料位置
1430.06 BOOL  ; 后上料伺服在原点位置
1430.09 BOOL  ; 后上料机构正常停止条件
1430.10 BOOL  ; 后上料机构清料停止条件
1430.15 BOOL  ; 后上料机构在设定位置
1431.00 BOOL  ; 后上料机构有错误
1431.01 BOOL  ; 后上料伺服手动定位目标位置设定OK
1431.02 BOOL  ; 后上料伺服自动定位目标位置设定OK
1431.03 BOOL  ; 后上料伺服到待机位条件
1431.04 BOOL  ; 后上料伺服到取料位条件
1431.05 BOOL  ; 后上料伺服到3#仓放料位安全条件
1431.06 BOOL  ; 后上料伺服到4#仓放料位安全条件
1431.07 BOOL  ; 后上料可向腔3
1431.08 BOOL  ; 后上料可向腔4
1435.00 BOOL  ; 后上料机构单次循环
1435.01 BOOL  ; 后上料机构单次循环完成
1435.02 BOOL  ; 后上料机构自动/单次循环
1436.00 BOOL  ; 后上料机构自动条件
1436.01 BOOL  ; 后上料机构步进条件
1436.15 BOOL  ; 后上料机构步进
1437 CHANNEL  ; 后上料自动步序
1437.00 BOOL  ; 后上料机构自动开始(步)
1437.01 BOOL  ; 后上料伺服到取料位(步)
1437.02 BOOL  ; 后上料升降气缸下降取料(步)
1437.03 BOOL  ; 后上料夹爪夹紧(步)
1437.04 BOOL  ; 后上料升降气缸取料后上升(步)
1437.05 BOOL  ; 后上料伺服到放料位&后进料旋转转回(步)
1437.06 BOOL  ; 后上料升降气缸下降放料(步)
1437.09 BOOL  ; 后上料夹爪松开(步)
1437.10 BOOL  ; 后上料升降气缸上升(步)
1437.11 BOOL  ; 后上料伺服到取料位(步)
1437.15 BOOL  ; 后上料自动运行结束(步)
143.00 BOOL  ; 出料伺服归零(M)
143.01 BOOL  ; 出料伺服点动前进(M)
143.02 BOOL  ; 出料伺服点动后退(M)
143.03 BOOL  ; 出料伺服到等待位置(M)
143.04 BOOL  ; 出料伺服到前取料位置(M)
143.05 BOOL  ; 出料伺服到后取料位置(M)
143.06 BOOL  ; 出料伺服到放料位置(M)
143.07 BOOL  ; 出料伺服到#2检测NG位置(M)
143.08 BOOL  ; 出料伺服到#3检测NG位置(M)
143.09 BOOL  ; 出料伺服到#4检测NG位置(M)
143.11 BOOL  ; 出料伺服手动定位条件
143.12 BOOL  ; 出料伺服手动定位(M)
143.13 BOOL  ; 出料伺服手动定位
143.15 BOOL  ; 出料机构复位(M)
1440.00 BOOL  ; 后下料机构在初始位
1440.01 BOOL  ; 后下料伺服在待机位置
1440.02 BOOL  ; 后下料伺服在仓3取料位置
1440.03 BOOL  ; 后下料伺服在仓4取料位置
1440.04 BOOL  ; 后下料伺服在放料位置
1440.05 BOOL  ; 后下料伺服在NG放料位置
1440.06 BOOL  ; 后下料伺服在原点位置
1440.07 BOOL  ; 下料3#NG放料位
1440.08 BOOL  ; 下料4#NG放料位
1440.09 BOOL  ; 后下料机构正常停止条件
1440.10 BOOL  ; 后下料机构清料停止条件
1440.15 BOOL  ; 后下料机构在设定位置
1441.00 BOOL  ; 后下料机构有错误
1441.01 BOOL  ; 后下料伺服手动定位目标位置设定OK
1441.02 BOOL  ; 后下料伺服自动定位目标位置设定OK
1441.03 BOOL  ; 后下料伺服到待机位条件
1441.04 BOOL  ; 后下料伺服到3#仓取料位条件
1441.05 BOOL  ; 后下料伺服到4#仓取料位安全条件
1441.06 BOOL  ; 后下料伺服到放料位条件
1441.07 BOOL  ; 后下料可向腔3
1441.08 BOOL  ; 后下料可向腔4
1445.00 BOOL  ; 后下料机构单次循环
1445.01 BOOL  ; 后下料机构单次循环完成
1445.02 BOOL  ; 后下料机构自动/单次循环
1446.00 BOOL  ; 后下料机构自动条件
1446.01 BOOL  ; 后下料机构步进条件
1446.15 BOOL  ; 后下料机构步进
1447 CHANNEL  ; 后下料自动步序
1447.00 BOOL  ; 后下料机构自动开始(步)
1447.01 BOOL  ; 后下料到取料位(步)
1447.02 BOOL  ; 后下料升降下降取料(步)
1447.03 BOOL  ; 后下料夹爪夹紧(步)
1447.05 BOOL  ; 后下料升降取料后上升(步)
1447.06 BOOL  ; 后下料伺服到放料位(步)
1447.07 BOOL  ; 后下料升降气缸下降放料(步)
1447.08 BOOL  ; 后下料请求
1447.09 BOOL  ; 后下料夹爪松开(步)
1447.10 BOOL  ; 后下料升降气缸放料后上升(步)
1447.11 BOOL  ; 后下料伺服到待机位(步)
1447.12 BOOL  ; 后旋转气缸旋转(步)
1447.14 BOOL  ; 后下料自动完成(步)
144.00 BOOL  ; 1真空泵启动(M)
144.01 BOOL  ; 1真空泵停止(M)
144.02 BOOL  ; #1吹气启动(M)
144.03 BOOL  ; #1吹气停止(M)
144.04 BOOL  ; 氦检仪启动(M)
144.05 BOOL  ; 氦检仪停止(M)
144.06 BOOL  ; #2吹气启动(M)
144.07 BOOL  ; #2吹气停止(M)
144.08 BOOL  ; #3吹气启动(M)
144.09 BOOL  ; #3吹气停止(M)
144.10 BOOL  ; #4吹气启动(M)
144.11 BOOL  ; #4吹气停止(M)
1450.00 BOOL  ; 1#腔体机构在初始位
1450.09 BOOL  ; 1#腔体机构正常停止条件
1450.10 BOOL  ; 1#腔体机构清料停止条件
1451.00 BOOL  ; 1#腔体机构有错误
1451.01 BOOL  ; 1#腔平移气缸运行安全条件
1451.10 BOOL  ; 1#腔体机构步自动步序错误
1455.00 BOOL  ; 1#腔体机构单次循环
1455.01 BOOL  ; 1#腔体机构单次循环完成
1455.02 BOOL  ; 1#腔体机构自动/单次循环
1456.00 BOOL  ; 1#腔体机构自动条件
1456.01 BOOL  ; 1#腔体机构步进条件
1456.15 BOOL  ; 1#腔体机构步进
1457 CHANNEL  ; 1#腔体自动步序
1457.00 BOOL  ; 1#腔体机构自动开始(步)
1457.01 BOOL  ; #1腔平移气缸后退(步)
1457.02 BOOL  ; #1腔顶升气缸上升(步)
1457.03 BOOL  ; #1腔密封气缸下降(步)
1457.04 BOOL  ; #1腔抽真空阀打开(步)
1457.05 BOOL  ; #1腔抽真空阀关闭(步)
1457.06 BOOL  ; #1腔氦检(步)
1457.07 BOOL  ; #1腔氦检结果判断(步)
1457.08 BOOL  ; #1腔氦检后抽残气(步)
1457.09 BOOL  ; #1腔氦检后破真空(步)
1457.10 BOOL  ; #1腔NG后清氦(步)
1457.11 BOOL  ; #1腔开模&密封气缸上升&吹气(步)
1457.12 BOOL  ; #1腔平移气缸前进&破真空阀关闭(步)
1457.13 BOOL  ; #1腔(步)
1457.14 BOOL  ; #1腔测试完成(步)
1457.15 BOOL  ; #1腔自动运行结束(步)
1459.08 BOOL  ; #1腔腔体抽气阀打开条件(A)
1459.10 BOOL  ; #1腔破真空条件
145.00 BOOL  ; #1腔平移气缸前进(M)
145.01 BOOL  ; #1腔平移气缸后退(M)
145.02 BOOL  ; #1腔顶升气缸上升(M)
145.03 BOOL  ; #1腔顶升气缸下降(M)
145.04 BOOL  ; #1腔密封气缸上升(M)
145.05 BOOL  ; #1腔密封气缸下降(M)
145.06 BOOL  ; #1腔电池抽气阀打开(M)
145.07 BOOL  ; #1腔电池抽气阀关闭(M)
145.08 BOOL  ; #1腔腔体抽气阀打开(M)
145.09 BOOL  ; #1腔腔体抽气阀关闭(M)
145.10 BOOL  ; #1腔电池破真空阀打开(M)
145.11 BOOL  ; #1腔电池破真空阀关闭(M)
145.12 BOOL  ; #1腔腔体破真空阀打开(M)
145.13 BOOL  ; #1腔腔体破真空阀关闭(M)
145.14 BOOL  ; #1腔注氦气阀打开(M)
145.15 BOOL  ; #1腔注氦气阀关闭(M)
1460.00 BOOL  ; 2#腔体机构在初始位
1460.09 BOOL  ; 2#腔体机构正常停止条件
1460.10 BOOL  ; 2#腔体机构清料停止条件
1461.00 BOOL  ; 2#腔体机构有错误
1461.01 BOOL  ; 2#腔平移气缸运行安全条件
1461.10 BOOL  ; 2#腔体机构步自动步序错误
1465.00 BOOL  ; 2#腔体机构单次循环
1465.01 BOOL  ; 2#腔体机构单次循环完成
1465.02 BOOL  ; 2#腔体机构自动/单次循环
1466.00 BOOL  ; 2#腔体机构自动条件
1466.01 BOOL  ; 2#腔体机构步进条件
1466.15 BOOL  ; 2#腔体机构步进
1467 CHANNEL  ; 2#腔体自动步序
1467.00 BOOL  ; 2#腔体机构自动开始(步)
1467.01 BOOL  ; 2#腔平移气缸后退(步)
1467.02 BOOL  ; 2#腔顶升气缸上升(步)
1467.03 BOOL  ; 2#腔密封气缸下降(步)
1467.04 BOOL  ; 2#腔抽真空阀打开(步)
1467.05 BOOL  ; 2#腔抽真空阀关闭(步)
1467.06 BOOL  ; 2#腔氦检(步)
1467.07 BOOL  ; 2#腔氦检结果判断(步)
1467.08 BOOL  ; 2#腔氦检后抽残气(步)
1467.09 BOOL  ; 2#腔氦检后破真空(步)
1467.10 BOOL  ; #2腔NG后清氦(步)
1467.11 BOOL  ; 2#腔开模&密封气缸上升&吹气(步)
1467.12 BOOL  ; 2#腔平移气缸前进&破真空阀关闭(步)
1467.13 BOOL  ; 2#腔(步)
1467.14 BOOL  ; 2#腔测试完成(步)
1467.15 BOOL  ; 2#腔自动运行结束(步)
1469.08 BOOL  ; #2腔腔体抽气阀打开条件(A)
1469.10 BOOL  ; #2模组电池破真空条件
146.00 BOOL  ; #1腔氦检阀打开(M)
146.01 BOOL  ; #1腔氦检阀关闭(M)
146.02 BOOL  ; #1腔腔体自检启动(M)
146.03 BOOL  ; #1腔腔体自检停止(M)
146.08 BOOL  ; 真空泵1启动
146.09 BOOL  ; 真空泵2启动
146.15 BOOL  ; #1腔机构复位(M)
1470.00 BOOL  ; 3#腔体机构在初始位
1470.09 BOOL  ; 3#腔体机构正常停止条件
1470.10 BOOL  ; 3#腔体机构清料停止条件
1471.00 BOOL  ; 3#腔体机构有错误
1471.01 BOOL  ; 3#腔平移气缸运行安全条件
1471.10 BOOL  ; 3#腔体机构步自动步序错误
1475.00 BOOL  ; 3#腔体机构单次循环
1475.01 BOOL  ; 3#腔体机构单次循环完成
1475.02 BOOL  ; 3#腔体机构自动/单次循环
1476.00 BOOL  ; 3#腔体机构自动条件
1476.01 BOOL  ; 3#腔体机构步进条件
1476.15 BOOL  ; 3#腔体机构步进
1477 CHANNEL  ; 3#腔体自动步序
1477.00 BOOL  ; 3#腔体机构自动开始(步)
1477.01 BOOL  ; 3#腔平移气缸后退(步)
1477.02 BOOL  ; 3#腔顶升气缸上升(步)
1477.03 BOOL  ; 3#腔密封气缸下降(步)
1477.04 BOOL  ; 3#腔抽真空阀打开(步)
1477.05 BOOL  ; 3#腔抽真空阀关闭(步)
1477.06 BOOL  ; 3#腔氦检(步)
1477.07 BOOL  ; 3#腔氦检结果判断(步)
1477.08 BOOL  ; 3#腔氦检后抽残气(步)
1477.09 BOOL  ; 3#腔氦检后破真空(步)
1477.10 BOOL  ; #3腔NG后清氦(步)
1477.11 BOOL  ; 3#腔开模&密封气缸上升&吹气(步)
1477.12 BOOL  ; 3#腔平移气缸前进&破真空阀关闭(步)
1477.13 BOOL  ; 3#腔(步)
1477.14 BOOL  ; 3#腔测试完成(步)
1477.15 BOOL  ; 3#腔自动运行结束(步)
1479.08 BOOL  ; #3腔腔体抽气阀打开条件(A)
1479.10 BOOL  ; #3腔电池破真空阀打开条件(A)
147.00 BOOL  ; #2腔平移气缸前进(M)
147.01 BOOL  ; #2腔平移气缸后退(M)
147.02 BOOL  ; #2腔顶升气缸上升(M)
147.03 BOOL  ; #2腔顶升气缸下降(M)
147.04 BOOL  ; #2腔密封气缸上升(M)
147.05 BOOL  ; #2腔密封气缸下降(M)
147.06 BOOL  ; #2腔电池抽气阀打开(M)
147.07 BOOL  ; #2腔电池抽气阀关闭(M)
147.08 BOOL  ; #2腔腔体抽气阀打开(M)
147.09 BOOL  ; #2腔腔体抽气阀关闭(M)
147.10 BOOL  ; #2腔电池破真空阀打开(M)
147.11 BOOL  ; #2腔电池破真空阀关闭(M)
147.12 BOOL  ; #2腔腔体破真空阀打开(M)
147.13 BOOL  ; #2腔腔体破真空阀关闭(M)
147.14 BOOL  ; #2腔注氦气阀打开(M)
147.15 BOOL  ; #2腔注氦气阀关闭(M)
1480.00 BOOL  ; 4#腔体机构在初始位
1480.02 BOOL  ; 出料升降伺服取料高度
1480.03 BOOL  ; 出料升降伺服放料高度
1480.09 BOOL  ; 4#腔体机构正常停止条件
1480.10 BOOL  ; 4#腔体机构清料停止条件
1481.00 BOOL  ; 4#腔体机构有错误
1481.01 BOOL  ; 4#腔平移气缸运行安全条件
1481.10 BOOL  ; 4#腔体机构步自动步序错误
1485.00 BOOL  ; 4#腔体机构单次循环
1485.01 BOOL  ; 4#腔体机构单次循环完成
1485.02 BOOL  ; 4#腔体机构自动/单次循环
1486.00 BOOL  ; 4#腔体机构自动条件
1486.01 BOOL  ; 4#腔体机构步进条件
1486.15 BOOL  ; 4#腔体机构步进
1487 CHANNEL  ; 4#腔体自动步序
1487.00 BOOL  ; 4#腔体机构自动开始(步)
1487.01 BOOL  ; 4#腔平移气缸后退(步)
1487.02 BOOL  ; 4#腔顶升气缸上升(步)
1487.03 BOOL  ; 4#腔密封气缸下降(步)
1487.04 BOOL  ; 4#腔抽真空阀打开(步)
1487.05 BOOL  ; 4#腔抽真空阀关闭(步)
1487.06 BOOL  ; 4#腔氦检(步)
1487.07 BOOL  ; 4#腔氦检结果判断(步)
1487.08 BOOL  ; 4#腔氦检后抽残气(步)
1487.09 BOOL  ; 4#腔氦检后破真空(步)
1487.10 BOOL  ; #4腔NG后清氦(步)
1487.11 BOOL  ; 4#腔开模&密封气缸上升&吹气(步)
1487.12 BOOL  ; 4#腔平移气缸前进&破真空阀关闭(步)
1487.13 BOOL  ; 4#腔(步)
1487.14 BOOL  ; 4#腔测试完成(步)
1487.15 BOOL  ; 4#腔自动运行结束(步)
1489.08 BOOL  ; #4腔腔体抽气阀打开条件(A)
1489.10 BOOL  ; #4模组电池破真空条件
148.00 BOOL  ; #2腔氦检阀打开(M)
148.01 BOOL  ; #2腔氦检阀关闭(M)
148.02 BOOL  ; #2腔腔体自检启动(M)
148.03 BOOL  ; #2腔腔体自检停止(M)
148.15 BOOL  ; #2腔机构复位(M)
1490.00 BOOL  ; 出料机构在初始位
1490.01 BOOL  ; 出料伺服在#1NG位置
1490.02 BOOL  ; 出料伺服在前取料位置
1490.03 BOOL  ; 出料伺服在后取料位置
1490.04 BOOL  ; 出料伺服在放料位置
1490.05 BOOL  ; 出料伺服在拉带安全位
1490.06 BOOL  ; 出料伺服在#2检测NG位
1490.07 BOOL  ; 下料3#NG放料位
1490.08 BOOL  ; 下料4#NG放料位
1490.09 BOOL  ; 出料机构正常停止条件
1490.10 BOOL  ; 出料机构清料停止条件
1490.11 BOOL  ; 出料伺服在后出料旋转安全位
1490.15 BOOL  ; 进料伺服在设定位置
1491.00 BOOL  ; 出料机构有错误
1491.01 BOOL  ; 出料伺服手动定位目标位置设定OK
1491.02 BOOL  ; 出料伺服自动定位目标位置设定OK
1491.03 BOOL  ; 出料伺服到待机位条件
1491.04 BOOL  ; 出料伺服到前取料位安全条件
1491.05 BOOL  ; 出料伺服到后取料位安全条件
1491.06 BOOL  ; 出料伺服到放料位安全条件
1491.10 BOOL  ; 出料伺服长距离定位
1495.00 BOOL  ; 出料机构单次循环
1495.01 BOOL  ; 出料机构单次循环完成
1495.02 BOOL  ; 出料机构自动/单次循环
1496.00 BOOL  ; 出料机构自动条件
1496.01 BOOL  ; 出料机构步进条件
1496.15 BOOL  ; 出料机构步进
1497 CHANNEL  ; 出料机构自动步序
1497.00 BOOL  ; 出料机构自动开始(步)
1497.01 BOOL  ; 到前|后取料位
1497.02 BOOL  ; 等待放料（步）
1497.03 BOOL  ; 等待气缸回升(步)
1497.04 BOOL  ; 出料到OK/NG位(步)
1497.05 BOOL  ; 出料升降取料后上升(步)
1497.06 BOOL  ; 出料归零(步)
1497.07 BOOL  ; 出料到待机位(步)
1497.08 BOOL  ; 循环结束(步)
1497.09 BOOL  ; 出料伺服到放料位&&出料平移张开(步)
1497.10 BOOL  ; 出料升降下降放料&出料旋转转回(步)
1497.11 BOOL  ; 出料夹爪松开放料(步)
1497.12 BOOL  ; 出料升降放料后上升(步)
1497.13 BOOL  ; 出料伺服到待机位&出料平移关闭(步)
1497.14 BOOL  ; 出料完成(步)
1499.00 BOOL  ; 出料升降气缸上升条件(A)
1499.04 BOOL  ; 出料平移气缸开条件(A)
1499.05 BOOL  ; 出料平移气缸合条件(A)
149.00 BOOL  ; #3腔平移气缸前进(M)
149.01 BOOL  ; #3腔平移气缸后退(M)
149.02 BOOL  ; #3腔顶升气缸上升(M)
149.03 BOOL  ; #3腔顶升气缸下降(M)
149.04 BOOL  ; #3腔密封气缸上升(M)
149.05 BOOL  ; #3腔密封气缸下降(M)
149.06 BOOL  ; #3腔电池抽气阀打开(M)
149.07 BOOL  ; #3腔电池抽气阀关闭(M)
149.08 BOOL  ; #3腔腔体抽气阀打开(M)
149.09 BOOL  ; #3腔腔体抽气阀关闭(M)
149.10 BOOL  ; #3腔电池破真空阀打开(M)
149.11 BOOL  ; #3腔电池破真空阀关闭(M)
149.12 BOOL  ; #3腔腔体破真空阀打开(M)
149.13 BOOL  ; #3腔腔体破真空阀关闭(M)
149.14 BOOL  ; #3腔注氦气阀打开(M)
149.15 BOOL  ; #3腔注氦气阀关闭(M)
14.00 BOOL  ; 进料升降伺服刹车
14.01 BOOL  ; 出料升降伺服刹车
14.02 BOOL  ; 取料可移动信号-拉带对接信号
14.03 BOOL  ; 放料可移动信号-拉带对接信号
14.04 BOOL  ; 故障信号-拉带对接信号
14.05 BOOL  ; 准备放料
14.06 BOOL  ; 取料准备信号-拉带对接信号
14.07 BOOL  ; nc
14.08 BOOL  ; #1腔体破真空阀
14.09 BOOL  ; #1电池破真空阀
14.10 BOOL  ; #2腔体抽气阀
14.11 BOOL  ; #2电池抽气阀
14.12 BOOL  ; #2电池注氦阀
14.13 BOOL  ; #2腔体氦检阀
14.14 BOOL  ; #2腔体破真空阀
14.15 BOOL  ; #2电池破真空阀
1509.15 BOOL  ; 端口1执行标志位
150.00 BOOL  ; #3腔氦检阀打开(M)
150.01 BOOL  ; #3腔氦检阀关闭(M)
150.02 BOOL  ; #3腔腔体自检启动(M)
150.03 BOOL  ; #3腔腔体自检停止(M)
150.15 BOOL  ; #3腔机构复位(M)
1519.15 BOOL  ; 端口2指令执行标志
151.00 BOOL  ; #4腔平移气缸前进(M)
151.01 BOOL  ; #4腔平移气缸后退(M)
151.02 BOOL  ; #4腔顶升气缸上升(M)
151.03 BOOL  ; #4腔顶升气缸下降(M)
151.04 BOOL  ; #4腔密封气缸上升(M)
151.05 BOOL  ; #4腔密封气缸下降(M)
151.06 BOOL  ; #4腔电池抽气阀打开(M)
151.07 BOOL  ; #4腔电池抽气阀关闭(M)
151.08 BOOL  ; #4腔腔体抽气阀打开(M)
151.09 BOOL  ; #4腔腔体抽气阀关闭(M)
151.10 BOOL  ; #4腔电池破真空阀打开(M)
151.11 BOOL  ; #4腔电池破真空阀关闭(M)
151.12 BOOL  ; #4腔腔体破真空阀打开(M)
151.13 BOOL  ; #4腔腔体破真空阀关闭(M)
151.14 BOOL  ; #4腔注氦气阀打开(M)
151.15 BOOL  ; #4腔注氦气阀关闭(M)
152.00 BOOL  ; #4腔氦检阀打开(M)
152.01 BOOL  ; #4腔氦检阀关闭(M)
152.02 BOOL  ; #4腔腔体自检启动(M)
152.03 BOOL  ; #4腔腔体自检停止(M)
152.15 BOOL  ; #4腔机构复位(M)
154.00 BOOL  ; 进料机械手升降气缸上升(复位)
154.01 BOOL  ; 进料机械手平移气缸合位(复位)
154.02 BOOL  ; 进料夹爪气缸张开(复位)
154.03 BOOL  ; 前腔体入料顶升气缸(复位)
154.04 BOOL  ; 后腔体入料顶升气缸(复位)
154.05 BOOL  ; 扫码NG缓存避位气缸后退(复位)(M)
154.06 BOOL  ; 扫码NG缓存接料气缸后退(复位)
154.07 BOOL  ; 扫码NG缓存间隔气缸上升复位)
154.08 BOOL  ; 进料夹爪气缸夹紧(复位)
154.09 BOOL  ; 进料伺服归零(复位)(M)
154.10 BOOL  ; 进料伺服到待机位置(复位)
154.12 BOOL  ; 扫码阻挡气缸前进(复位)(M)
155.00 BOOL  ; 腔体1电池密封气缸上升(复位)
155.01 BOOL  ; 腔体1顶升气缸下降(复位)
155.02 BOOL  ; 腔体1平移气缸前进(复位)
155.03 BOOL  ; 腔体1腔体破真空(复位)
155.04 BOOL  ; 腔体1电池破真空(复位)
156.00 BOOL  ; 腔体2电池密封气缸上升(复位)
156.01 BOOL  ; 腔体2顶升气缸下降(复位)
156.02 BOOL  ; 腔体2平移气缸前进(复位)
156.03 BOOL  ; 腔体2腔体破真空(复位)
156.04 BOOL  ; 腔体2电池破真空(复位)
1575.00 BOOL  ; SCU21_3 Port#1 Wait Release Switch
1575.01 BOOL  ; SCU21_3 Port#1 Continuous Trace Switch
1575.02 BOOL  ; SCU21_3 Port#1 One-shot Trace Switch
1575.03 BOOL  ; SCU21_3 Port#1 Abort Switch
1575.04 BOOL  ; SCU21_3 Port#1 Serial Gateway Prohibited Switch
1575.05 BOOL  ; SCU21_3 Port#1 Reserved
1575.06 BOOL  ; SCU21_3 Port#1 Loopback Test Switch
1575.07 BOOL  ; SCU21_3 Port#1 Reserved
1575.08 BOOL  ; SCU21_3 Port#2 Wait Release Switch
1575.09 BOOL  ; SCU21_3 Port#2 Continuous Trace Switch
1575.10 BOOL  ; SCU21_3 Port#2 One-shot Trace Switch
1575.11 BOOL  ; SCU21_3 Port#2 Abort Switch
1575.12 BOOL  ; SCU21_3 Port#2 Serial Gateway Prohibited Switch
1575.13 BOOL  ; SCU21_3 Port#2 Reserved
1575.14 BOOL  ; SCU21_3 Port#2 Loopback Test Switch
1575.15 BOOL  ; SCU21_3 Port#2 Reserved
1576.00 BOOL  ; SCU21_3 Protocol Data Error
1576.01 BOOL  ; SCU21_3 Error Log EEPROM Error
1576.02 BOOL  ; SCU21_3 Reserved
1576.03 BOOL  ; SCU21_3 Reserved
1576.04 BOOL  ; SCU21_3 Reserved
1576.05 BOOL  ; SCU21_3 Reserved
1576.06 BOOL  ; SCU21_3 Reserved
1576.07 BOOL  ; SCU21_3 Reserved
1576.08 BOOL  ; SCU21_3 Reserved
1576.09 BOOL  ; SCU21_3 Reserved
1576.10 BOOL  ; SCU21_3 Reserved
1576.11 BOOL  ; SCU21_3 Reserved
1576.12 BOOL  ; SCU21_3 Reserved
1576.13 BOOL  ; SCU21_3 Reserved
1576.14 BOOL  ; SCU21_3 Reserved
1576.15 BOOL  ; SCU21_3 Reserved
1577.00 BOOL  ; SCU21_3 Reserved
1577.01 BOOL  ; SCU21_3 Reserved
1577.02 BOOL  ; SCU21_3 Reserved
1577.03 BOOL  ; SCU21_3 Reserved
1577.04 BOOL  ; SCU21_3 Reserved
1577.05 BOOL  ; SCU21_3 Reserved
1577.06 BOOL  ; SCU21_3 Reserved
1577.07 BOOL  ; SCU21_3 Reserved
1577.08 BOOL  ; SCU21_3 Reserved
1577.09 BOOL  ; SCU21_3 Reserved
1577.10 BOOL  ; SCU21_3 Reserved
1577.11 BOOL  ; SCU21_3 Reserved
1577.12 BOOL  ; SCU21_3 Reserved
1577.13 BOOL  ; SCU21_3 Reserved
1577.14 BOOL  ; SCU21_3 Reserved
1577.15 BOOL  ; SCU21_3 Reserved
1578.00 BOOL  ; SCU21_3 Reserved
1578.01 BOOL  ; SCU21_3 Reserved
1578.02 BOOL  ; SCU21_3 Reserved
1578.03 BOOL  ; SCU21_3 Reserved
1578.04 BOOL  ; SCU21_3 Reserved
1578.05 BOOL  ; SCU21_3 Reserved
1578.06 BOOL  ; SCU21_3 Reserved
1578.07 BOOL  ; SCU21_3 Reserved
1578.08 BOOL  ; SCU21_3 Reserved
1578.09 BOOL  ; SCU21_3 Reserved
1578.10 BOOL  ; SCU21_3 Reserved
1578.11 BOOL  ; SCU21_3 Reserved
1578.12 BOOL  ; SCU21_3 Reserved
1578.13 BOOL  ; SCU21_3 Reserved
1578.14 BOOL  ; SCU21_3 Reserved
1578.15 BOOL  ; SCU21_3 Reserved
1579.00 BOOL  ; SCU21_3 Reserved
1579.01 BOOL  ; SCU21_3 Reserved
1579.02 BOOL  ; SCU21_3 Reserved
1579.03 BOOL  ; SCU21_3 Reserved
1579.04 BOOL  ; SCU21_3 Reserved
1579.05 BOOL  ; SCU21_3 Reserved
1579.06 BOOL  ; SCU21_3 Reserved
1579.07 BOOL  ; SCU21_3 Reserved
1579.08 BOOL  ; SCU21_3 Reserved
1579.09 BOOL  ; SCU21_3 Reserved
1579.10 BOOL  ; SCU21_3 Reserved
1579.11 BOOL  ; SCU21_3 Reserved
1579.12 BOOL  ; SCU21_3 Reserved
1579.13 BOOL  ; SCU21_3 Reserved
1579.14 BOOL  ; SCU21_3 Reserved
1579.15 BOOL  ; SCU21_3 Reserved
157.00 BOOL  ; 腔体3电池密封气缸上升(复位)
157.01 BOOL  ; 腔体3顶升气缸下降(复位)
157.02 BOOL  ; 腔体3平移气缸前进(复位)
157.03 BOOL  ; 腔体3腔体破真空(复位)
157.04 BOOL  ; 腔体3电池破真空(复位)
1580.00 BOOL  ; SCU21_3 Port#1 Parity: Even/Odd
1580.01 BOOL  ; SCU21_3 Port#1 Parity: Yes/No
1580.02 BOOL  ; SCU21_3 Port#1 Stop bits: 1 or 2 bits
1580.03 BOOL  ; SCU21_3 Port#1 Data length: 7 or 8 bits
1580.04 BOOL  ; SCU21_3 Port#1 Start bits: Always 1
1580.05 BOOL  ; SCU21_3 Port#1 Reserved
1580.06 BOOL  ; SCU21_3 Port#1 Reserved
1580.07 BOOL  ; SCU21_3 Port#1 Reserved
1580.08 BOOL  ; SCU21_3 Port#1 Baud rate
1580.09 BOOL  ; SCU21_3 Port#1 Baud rate
1580.10 BOOL  ; SCU21_3 Port#1 Baud rate
1580.11 BOOL  ; SCU21_3 Port#1 Baud rate
1580.12 BOOL  ; SCU21_3 Port#1 Serial communications mode
1580.13 BOOL  ; SCU21_3 Port#1 Serial communications mode
1580.14 BOOL  ; SCU21_3 Port#1 Serial communications mode
1580.15 BOOL  ; SCU21_3 Port#1 Serial communications mode
1581.00 BOOL  ; SCU21_3 Port#1 1: Port operating; 0: Port stopped
1581.01 BOOL  ; SCU21_3 Port#1 1: System Setup error; 0: System Setup normal
1581.02 BOOL  ; SCU21_3 Port#1 Reserved
1581.03 BOOL  ; SCU21_3 Port#1 Reserved
1581.04 BOOL  ; SCU21_3 Port#1 Reserved
1581.05 BOOL  ; SCU21_3 Port#1 Reserved
1581.06 BOOL  ; SCU21_3 Port#1 Reserved
1581.07 BOOL  ; SCU21_3 Port#1 Reserved
1581.08 BOOL  ; SCU21_3 Port#1 Reserved
1581.09 BOOL  ; SCU21_3 Port#1 Reserved
1581.10 BOOL  ; SCU21_3 Port#1 Reserved
1581.11 BOOL  ; SCU21_3 Port#1 Reserved
1581.12 BOOL  ; SCU21_3 Port#1 Reserved
1581.13 BOOL  ; SCU21_3 Port#1 Terminating resistance
1581.14 BOOL  ; SCU21_3 Port#1 Hardware settings
1581.15 BOOL  ; SCU21_3 Port#1 Hardware settings
1582.00 BOOL  ; SCU21_3 Port#1 Reserved
1582.01 BOOL  ; SCU21_3 Port#1 Reserved
1582.02 BOOL  ; SCU21_3 Port#1 Reserved
1582.03 BOOL  ; SCU21_3 Port#1 RTS (RS) signal
1582.04 BOOL  ; SCU21_3 Port#1 CTS (CS) signal
1582.05 BOOL  ; SCU21_3 Port#1 Reserved
1582.06 BOOL  ; SCU21_3 Port#1 DSR (DR) signal
1582.07 BOOL  ; SCU21_3 Port#1 DTR (ER) signal
1582.08 BOOL  ; SCU21_3 Port#1 Local Unit busy receiving (Flow control)
1582.09 BOOL  ; SCU21_3 Port#1 Reserved
1582.10 BOOL  ; SCU21_3 Port#1 Remote Unit busy receiving (Flow control)
1582.11 BOOL  ; SCU21_3 Port#1 Reserved
1582.12 BOOL  ; SCU21_3 Port#1 Reserved
1582.13 BOOL  ; SCU21_3 Port#1 Reserved
1582.14 BOOL  ; SCU21_3 Port#1 Reserved
1582.15 BOOL  ; SCU21_3 Port#1 Reserved
1583.00 BOOL  ; SCU21_3 Port#1 Reserved
1583.01 BOOL  ; SCU21_3 Port#1 Reserved
1583.02 BOOL  ; SCU21_3 Port#1 Parity error
1583.03 BOOL  ; SCU21_3 Port#1 Framing error
1583.04 BOOL  ; SCU21_3 Port#1 Overrun error
1583.05 BOOL  ; SCU21_3 Port#1 Timeout error
1583.06 BOOL  ; SCU21_3 Port#1 Command error
1583.07 BOOL  ; SCU21_3 Port#1 FCS check error
1583.08 BOOL  ; SCU21_3 Port#1 Number of retries
1583.09 BOOL  ; SCU21_3 Port#1 Number of retries
1583.10 BOOL  ; SCU21_3 Port#1 Number of retries
1583.11 BOOL  ; SCU21_3 Port#1 Number of retries
1583.12 BOOL  ; SCU21_3 Port#1 Tr exceeded
1583.13 BOOL  ; SCU21_3 Port#1 Tfr exceeded
1583.14 BOOL  ; SCU21_3 Port#1 Tfs exceeded
1583.15 BOOL  ; SCU21_3 Port#1 Transmission error
1584.00 BOOL  ; SCU21_3 Port#1 Protocol status
1584.01 BOOL  ; SCU21_3 Port#1 Error codes
1584.02 BOOL  ; SCU21_3 Port#1 Error codes
1584.03 BOOL  ; SCU21_3 Port#1 Error codes
1584.04 BOOL  ; SCU21_3 Port#1 Reserved
1584.05 BOOL  ; SCU21_3 Port#1 Reserved
1584.06 BOOL  ; SCU21_3 Port#1 Reserved
1584.07 BOOL  ; SCU21_3 Port#1 Reserved
1584.08 BOOL  ; SCU21_3 Port#1 Serial Gateway Prohibited Flag
1584.09 BOOL  ; SCU21_3 Port#1 Sequence Waiting Flag
1584.10 BOOL  ; SCU21_3 Port#1 Sequence Abort Completion Flag
1584.11 BOOL  ; SCU21_3 Port#1 Sequence End Completion Flag
1584.12 BOOL  ; SCU21_3 Port#1 Tracing Flag
1584.13 BOOL  ; SCU21_3 Port#1 Aborted Flag
1584.14 BOOL  ; SCU21_3 Port#1 Step Troubleshooting Flag
1584.15 BOOL  ; SCU21_3 Port#1 Protocol Macro Executing Flag
1585.00 BOOL  ; SCU21_3 Port#1 Communications Sequence Number
1585.01 BOOL  ; SCU21_3 Port#1 Communications Sequence Number
1585.02 BOOL  ; SCU21_3 Port#1 Communications Sequence Number
1585.03 BOOL  ; SCU21_3 Port#1 Communications Sequence Number
1585.04 BOOL  ; SCU21_3 Port#1 Communications Sequence Number
1585.05 BOOL  ; SCU21_3 Port#1 Communications Sequence Number
1585.06 BOOL  ; SCU21_3 Port#1 Communications Sequence Number
1585.07 BOOL  ; SCU21_3 Port#1 Communications Sequence Number
1585.08 BOOL  ; SCU21_3 Port#1 Communications Sequence Number
1585.09 BOOL  ; SCU21_3 Port#1 Communications Sequence Number
1585.10 BOOL  ; SCU21_3 Port#1 Communications Sequence Number
1585.11 BOOL  ; SCU21_3 Port#1 Communications Sequence Number
1585.12 BOOL  ; SCU21_3 Port#1 Reserved
1585.13 BOOL  ; SCU21_3 Port#1 Reserved
1585.14 BOOL  ; SCU21_3 Port#1 Reserved
1585.15 BOOL  ; SCU21_3 Port#1 Reserved
1586.00 BOOL  ; SCU21_3 Port#1 Executed Reception Case Number
1586.01 BOOL  ; SCU21_3 Port#1 Executed Reception Case Number
1586.02 BOOL  ; SCU21_3 Port#1 Executed Reception Case Number
1586.03 BOOL  ; SCU21_3 Port#1 Executed Reception Case Number
1586.04 BOOL  ; SCU21_3 Port#1 Reserved
1586.05 BOOL  ; SCU21_3 Port#1 Reserved
1586.06 BOOL  ; SCU21_3 Port#1 Reserved
1586.07 BOOL  ; SCU21_3 Port#1 Reserved
1586.08 BOOL  ; SCU21_3 Port#1 Executed Step Number
1586.09 BOOL  ; SCU21_3 Port#1 Executed Step Number
1586.10 BOOL  ; SCU21_3 Port#1 Executed Step Number
1586.11 BOOL  ; SCU21_3 Port#1 Executed Step Number
1586.12 BOOL  ; SCU21_3 Port#1 Reserved
1586.13 BOOL  ; SCU21_3 Port#1 Reserved
1586.14 BOOL  ; SCU21_3 Port#1 Reserved
1586.15 BOOL  ; SCU21_3 Port#1 Reserved
1587.00 BOOL  ; SCU21_3 Port#1 Executed Reception Case Number Storage Flag
1587.01 BOOL  ; SCU21_3 Port#1 Executed Reception Case Number Storage Flag
1587.02 BOOL  ; SCU21_3 Port#1 Executed Reception Case Number Storage Flag
1587.03 BOOL  ; SCU21_3 Port#1 Executed Reception Case Number Storage Flag
1587.04 BOOL  ; SCU21_3 Port#1 Executed Reception Case Number Storage Flag
1587.05 BOOL  ; SCU21_3 Port#1 Executed Reception Case Number Storage Flag
1587.06 BOOL  ; SCU21_3 Port#1 Executed Reception Case Number Storage Flag
1587.07 BOOL  ; SCU21_3 Port#1 Executed Reception Case Number Storage Flag
1587.08 BOOL  ; SCU21_3 Port#1 Executed Reception Case Number Storage Flag
1587.09 BOOL  ; SCU21_3 Port#1 Executed Reception Case Number Storage Flag
1587.10 BOOL  ; SCU21_3 Port#1 Executed Reception Case Number Storage Flag
1587.11 BOOL  ; SCU21_3 Port#1 Executed Reception Case Number Storage Flag
1587.12 BOOL  ; SCU21_3 Port#1 Executed Reception Case Number Storage Flag
1587.13 BOOL  ; SCU21_3 Port#1 Executed Reception Case Number Storage Flag
1587.14 BOOL  ; SCU21_3 Port#1 Executed Reception Case Number Storage Flag
1587.15 BOOL  ; SCU21_3 Port#1 Executed Reception Case Number Storage Flag
1588.00 BOOL  ; SCU21_3 Port#1 Executed Step Number Storage Flag
1588.01 BOOL  ; SCU21_3 Port#1 Executed Step Number Storage Flag
1588.02 BOOL  ; SCU21_3 Port#1 Executed Step Number Storage Flag
1588.03 BOOL  ; SCU21_3 Port#1 Executed Step Number Storage Flag
1588.04 BOOL  ; SCU21_3 Port#1 Executed Step Number Storage Flag
1588.05 BOOL  ; SCU21_3 Port#1 Executed Step Number Storage Flag
1588.06 BOOL  ; SCU21_3 Port#1 Executed Step Number Storage Flag
1588.07 BOOL  ; SCU21_3 Port#1 Executed Step Number Storage Flag
1588.08 BOOL  ; SCU21_3 Port#1 Executed Step Number Storage Flag
1588.09 BOOL  ; SCU21_3 Port#1 Executed Step Number Storage Flag
1588.10 BOOL  ; SCU21_3 Port#1 Executed Step Number Storage Flag
1588.11 BOOL  ; SCU21_3 Port#1 Executed Step Number Storage Flag
1588.12 BOOL  ; SCU21_3 Port#1 Executed Step Number Storage Flag
1588.13 BOOL  ; SCU21_3 Port#1 Executed Step Number Storage Flag
1588.14 BOOL  ; SCU21_3 Port#1 Executed Step Number Storage Flag
1588.15 BOOL  ; SCU21_3 Port#1 Executed Step Number Storage Flag
1589.00 BOOL  ; SCU21_3 Port#1 Repeat Counter Present Value
1589.01 BOOL  ; SCU21_3 Port#1 Repeat Counter Present Value
1589.02 BOOL  ; SCU21_3 Port#1 Repeat Counter Present Value
1589.03 BOOL  ; SCU21_3 Port#1 Repeat Counter Present Value
1589.04 BOOL  ; SCU21_3 Port#1 Repeat Counter Present Value
1589.05 BOOL  ; SCU21_3 Port#1 Repeat Counter Present Value
1589.06 BOOL  ; SCU21_3 Port#1 Repeat Counter Present Value
1589.07 BOOL  ; SCU21_3 Port#1 Repeat Counter Present Value
1589.08 BOOL  ; SCU21_3 Port#1 Repeat Counter Setting Value
1589.09 BOOL  ; SCU21_3 Port#1 Repeat Counter Setting Value
1589.10 BOOL  ; SCU21_3 Port#1 Repeat Counter Setting Value
1589.11 BOOL  ; SCU21_3 Port#1 Repeat Counter Setting Value
1589.12 BOOL  ; SCU21_3 Port#1 Repeat Counter Setting Value
1589.13 BOOL  ; SCU21_3 Port#1 Repeat Counter Setting Value
1589.14 BOOL  ; SCU21_3 Port#1 Repeat Counter Setting Value
1589.15 BOOL  ; SCU21_3 Port#1 Repeat Counter Setting Value
158.00 BOOL  ; 腔体4电池密封气缸上升(复位)
158.01 BOOL  ; 腔体4顶升气缸下降(复位)
158.02 BOOL  ; 腔体4平移气缸前进(复位)
158.03 BOOL  ; 腔体4腔体破真空(复位)
158.04 BOOL  ; 腔体4电池破真空(复位)
1590.00 BOOL  ; SCU21_3 Port#2 Parity: Even/Odd
1590.01 BOOL  ; SCU21_3 Port#2 Parity: Yes/No
1590.02 BOOL  ; SCU21_3 Port#2 Stop bits: 1 or 2 bits
1590.03 BOOL  ; SCU21_3 Port#2 Data length: 7 or 8 bits
1590.04 BOOL  ; SCU21_3 Port#2 Start bits: Always 1
1590.05 BOOL  ; SCU21_3 Port#2 Reserved
1590.06 BOOL  ; SCU21_3 Port#2 Reserved
1590.07 BOOL  ; SCU21_3 Port#2 Reserved
1590.08 BOOL  ; SCU21_3 Port#2 Baud rate
1590.09 BOOL  ; SCU21_3 Port#2 Baud rate
1590.10 BOOL  ; SCU21_3 Port#2 Baud rate
1590.11 BOOL  ; SCU21_3 Port#2 Baud rate
1590.12 BOOL  ; SCU21_3 Port#2 Serial communications mode
1590.13 BOOL  ; SCU21_3 Port#2 Serial communications mode
1590.14 BOOL  ; SCU21_3 Port#2 Serial communications mode
1590.15 BOOL  ; SCU21_3 Port#2 Serial communications mode
1591.00 BOOL  ; SCU21_3 Port#2 1: Port operating; 0: Port stopped
1591.01 BOOL  ; SCU21_3 Port#2 1: System Setup error; 0: System Setup normal
1591.02 BOOL  ; SCU21_3 Port#2 Reserved
1591.03 BOOL  ; SCU21_3 Port#2 Reserved
1591.04 BOOL  ; SCU21_3 Port#2 Reserved
1591.05 BOOL  ; SCU21_3 Port#2 Reserved
1591.06 BOOL  ; SCU21_3 Port#2 Reserved
1591.07 BOOL  ; SCU21_3 Port#2 Reserved
1591.08 BOOL  ; SCU21_3 Port#2 Reserved
1591.09 BOOL  ; SCU21_3 Port#2 Reserved
1591.10 BOOL  ; SCU21_3 Port#2 Reserved
1591.11 BOOL  ; SCU21_3 Port#2 Reserved
1591.12 BOOL  ; SCU21_3 Port#2 Reserved
1591.13 BOOL  ; SCU21_3 Port#2 Terminating resistance
1591.14 BOOL  ; SCU21_3 Port#2 Hardware settings
1591.15 BOOL  ; SCU21_3 Port#2 Hardware settings
1592.00 BOOL  ; SCU21_3 Port#2 Reserved
1592.01 BOOL  ; SCU21_3 Port#2 Reserved
1592.02 BOOL  ; SCU21_3 Port#2 Reserved
1592.03 BOOL  ; SCU21_3 Port#2 RTS (RS) signal
1592.04 BOOL  ; SCU21_3 Port#2 CTS (CS) signal
1592.05 BOOL  ; SCU21_3 Port#2 Reserved
1592.06 BOOL  ; SCU21_3 Port#2 DSR (DR) signal
1592.07 BOOL  ; SCU21_3 Port#2 DTR (ER) signal
1592.08 BOOL  ; SCU21_3 Port#2 Local Unit busy receiving (Flow control)
1592.09 BOOL  ; SCU21_3 Port#2 Reserved
1592.10 BOOL  ; SCU21_3 Port#2 Remote Unit busy receiving (Flow control)
1592.11 BOOL  ; SCU21_3 Port#2 Reserved
1592.12 BOOL  ; SCU21_3 Port#2 Reserved
1592.13 BOOL  ; SCU21_3 Port#2 Reserved
1592.14 BOOL  ; SCU21_3 Port#2 Reserved
1592.15 BOOL  ; SCU21_3 Port#2 Reserved
1593.00 BOOL  ; SCU21_3 Port#2 Reserved
1593.01 BOOL  ; SCU21_3 Port#2 Reserved
1593.02 BOOL  ; SCU21_3 Port#2 Parity error
1593.03 BOOL  ; SCU21_3 Port#2 Framing error
1593.04 BOOL  ; SCU21_3 Port#2 Overrun error
1593.05 BOOL  ; SCU21_3 Port#2 Timeout error
1593.06 BOOL  ; SCU21_3 Port#2 Command error
1593.07 BOOL  ; SCU21_3 Port#2 FCS check error
1593.08 BOOL  ; SCU21_3 Port#2 Number of retries
1593.09 BOOL  ; SCU21_3 Port#2 Number of retries
1593.10 BOOL  ; SCU21_3 Port#2 Number of retries
1593.11 BOOL  ; SCU21_3 Port#2 Number of retries
1593.12 BOOL  ; SCU21_3 Port#2 Tr exceeded
1593.13 BOOL  ; SCU21_3 Port#2 Tfr exceeded
1593.14 BOOL  ; SCU21_3 Port#2 Tfs exceeded
1593.15 BOOL  ; SCU21_3 Port#2 Transmission error
1594.00 BOOL  ; SCU21_3 Port#2 Protocol status
1594.01 BOOL  ; SCU21_3 Port#2 Error codes
1594.02 BOOL  ; SCU21_3 Port#2 Error codes
1594.03 BOOL  ; SCU21_3 Port#2 Error codes
1594.04 BOOL  ; SCU21_3 Port#2 Reserved
1594.05 BOOL  ; SCU21_3 Port#2 Reserved
1594.06 BOOL  ; SCU21_3 Port#2 Reserved
1594.07 BOOL  ; SCU21_3 Port#2 Reserved
1594.08 BOOL  ; SCU21_3 Port#2 Serial Gateway Prohibited Flag
1594.09 BOOL  ; SCU21_3 Port#2 Sequence Waiting Flag
1594.10 BOOL  ; SCU21_3 Port#2 Sequence Abort Completion Flag
1594.11 BOOL  ; SCU21_3 Port#2 Sequence End Completion Flag
1594.12 BOOL  ; SCU21_3 Port#2 Tracing Flag
1594.13 BOOL  ; SCU21_3 Port#2 Aborted Flag
1594.14 BOOL  ; SCU21_3 Port#2 Step Troubleshooting Flag
1594.15 BOOL  ; SCU21_Port#2
1595.00 BOOL  ; SCU21_3 Port#2 Communications Sequence Number
1595.01 BOOL  ; SCU21_3 Port#2 Communications Sequence Number
1595.02 BOOL  ; SCU21_3 Port#2 Communications Sequence Number
1595.03 BOOL  ; SCU21_3 Port#2 Communications Sequence Number
1595.04 BOOL  ; SCU21_3 Port#2 Communications Sequence Number
1595.05 BOOL  ; SCU21_3 Port#2 Communications Sequence Number
1595.06 BOOL  ; SCU21_3 Port#2 Communications Sequence Number
1595.07 BOOL  ; SCU21_3 Port#2 Communications Sequence Number
1595.08 BOOL  ; SCU21_3 Port#2 Communications Sequence Number
1595.09 BOOL  ; SCU21_3 Port#2 Communications Sequence Number
1595.10 BOOL  ; SCU21_3 Port#2 Communications Sequence Number
1595.11 BOOL  ; SCU21_3 Port#2 Communications Sequence Number
1595.12 BOOL  ; SCU21_3 Port#2 Reserved
1595.13 BOOL  ; SCU21_3 Port#2 Reserved
1595.14 BOOL  ; SCU21_3 Port#2 Reserved
1595.15 BOOL  ; SCU21_3 Port#2 Reserved
1596.00 BOOL  ; SCU21_3 Port#2 Executed Reception Case Number
1596.01 BOOL  ; SCU21_3 Port#2 Executed Reception Case Number
1596.02 BOOL  ; SCU21_3 Port#2 Executed Reception Case Number
1596.03 BOOL  ; SCU21_3 Port#2 Executed Reception Case Number
1596.04 BOOL  ; SCU21_3 Port#2 Reserved
1596.05 BOOL  ; SCU21_3 Port#2 Reserved
1596.06 BOOL  ; SCU21_3 Port#2 Reserved
1596.07 BOOL  ; SCU21_3 Port#2 Reserved
1596.08 BOOL  ; SCU21_3 Port#2 Executed Step Number
1596.09 BOOL  ; SCU21_3 Port#2 Executed Step Number
1596.10 BOOL  ; SCU21_3 Port#2 Executed Step Number
1596.11 BOOL  ; SCU21_3 Port#2 Executed Step Number
1596.12 BOOL  ; SCU21_3 Port#2 Reserved
1596.13 BOOL  ; SCU21_3 Port#2 Reserved
1596.14 BOOL  ; SCU21_3 Port#2 Reserved
1596.15 BOOL  ; SCU21_3 Port#2 Reserved
1597.00 BOOL  ; SCU21_3 Port#2 Executed Reception Case Number Storage Flag
1597.01 BOOL  ; SCU21_3 Port#2 Executed Reception Case Number Storage Flag
1597.02 BOOL  ; SCU21_3 Port#2 Executed Reception Case Number Storage Flag
1597.03 BOOL  ; SCU21_3 Port#2 Executed Reception Case Number Storage Flag
1597.04 BOOL  ; SCU21_3 Port#2 Executed Reception Case Number Storage Flag
1597.05 BOOL  ; SCU21_3 Port#2 Executed Reception Case Number Storage Flag
1597.06 BOOL  ; SCU21_3 Port#2 Executed Reception Case Number Storage Flag
1597.07 BOOL  ; SCU21_3 Port#2 Executed Reception Case Number Storage Flag
1597.08 BOOL  ; SCU21_3 Port#2 Executed Reception Case Number Storage Flag
1597.09 BOOL  ; SCU21_3 Port#2 Executed Reception Case Number Storage Flag
1597.10 BOOL  ; SCU21_3 Port#2 Executed Reception Case Number Storage Flag
1597.11 BOOL  ; SCU21_3 Port#2 Executed Reception Case Number Storage Flag
1597.12 BOOL  ; SCU21_3 Port#2 Executed Reception Case Number Storage Flag
1597.13 BOOL  ; SCU21_3 Port#2 Executed Reception Case Number Storage Flag
1597.14 BOOL  ; SCU21_3 Port#2 Executed Reception Case Number Storage Flag
1597.15 BOOL  ; SCU21_3 Port#2 Executed Reception Case Number Storage Flag
1598.00 BOOL  ; SCU21_3 Port#2 Executed Step Number Storage Flag
1598.01 BOOL  ; SCU21_3 Port#2 Executed Step Number Storage Flag
1598.02 BOOL  ; SCU21_3 Port#2 Executed Step Number Storage Flag
1598.03 BOOL  ; SCU21_3 Port#2 Executed Step Number Storage Flag
1598.04 BOOL  ; SCU21_3 Port#2 Executed Step Number Storage Flag
1598.05 BOOL  ; SCU21_3 Port#2 Executed Step Number Storage Flag
1598.06 BOOL  ; SCU21_3 Port#2 Executed Step Number Storage Flag
1598.07 BOOL  ; SCU21_3 Port#2 Executed Step Number Storage Flag
1598.08 BOOL  ; SCU21_3 Port#2 Executed Step Number Storage Flag
1598.09 BOOL  ; SCU21_3 Port#2 Executed Step Number Storage Flag
1598.10 BOOL  ; SCU21_3 Port#2 Executed Step Number Storage Flag
1598.11 BOOL  ; SCU21_3 Port#2 Executed Step Number Storage Flag
1598.12 BOOL  ; SCU21_3 Port#2 Executed Step Number Storage Flag
1598.13 BOOL  ; SCU21_3 Port#2 Executed Step Number Storage Flag
1598.14 BOOL  ; SCU21_3 Port#2 Executed Step Number Storage Flag
1598.15 BOOL  ; SCU21_3 Port#2 Executed Step Number Storage Flag
1599.00 BOOL  ; SCU21_3 Port#2 Repeat Counter Present Value
1599.01 BOOL  ; SCU21_3 Port#2 Repeat Counter Present Value
1599.02 BOOL  ; SCU21_3 Port#2 Repeat Counter Present Value
1599.03 BOOL  ; SCU21_3 Port#2 Repeat Counter Present Value
1599.04 BOOL  ; SCU21_3 Port#2 Repeat Counter Present Value
1599.05 BOOL  ; SCU21_3 Port#2 Repeat Counter Present Value
1599.06 BOOL  ; SCU21_3 Port#2 Repeat Counter Present Value
1599.07 BOOL  ; SCU21_3 Port#2 Repeat Counter Present Value
1599.08 BOOL  ; SCU21_3 Port#2 Repeat Counter Setting Value
1599.09 BOOL  ; SCU21_3 Port#2 Repeat Counter Setting Value
1599.10 BOOL  ; SCU21_3 Port#2 Repeat Counter Setting Value
1599.11 BOOL  ; SCU21_3 Port#2 Repeat Counter Setting Value
1599.12 BOOL  ; SCU21_3 Port#2 Repeat Counter Setting Value
1599.13 BOOL  ; SCU21_3 Port#2 Repeat Counter Setting Value
1599.14 BOOL  ; SCU21_3 Port#2 Repeat Counter Setting Value
1599.15 BOOL  ; SCU21_3 Port#2 Repeat Counter Setting Value
159.00 BOOL  ; 出料机械手升降气缸上升(复位)
159.01 BOOL  ; 出料机械手平移气缸合(复位)
159.02 BOOL  ; 出料夹爪气缸张开(复位)
159.03 BOOL  ; #1测试NG气缸(复位)
159.04 BOOL  ; #2测试NG气缸(复位)
159.05 BOOL  ; 前腔体出料顶升气缸(复位)
159.06 BOOL  ; 后腔体出料顶升气缸(复位)
159.07 BOOL  ; 出料夹爪气缸夹紧(复位)
159.09 BOOL  ; 出料伺服归零(复位)(M)
159.10 BOOL  ; 出料伺服到待机位置(复位)
15.00 BOOL  ; #3腔体抽气阀
15.01 BOOL  ; #3电池抽气阀
15.02 BOOL  ; #3电池注氦阀
15.03 BOOL  ; #3腔体氦检阀
15.04 BOOL  ; #3腔体破真空阀
15.05 BOOL  ; #3电池破真空阀
15.06 BOOL  ; #4腔体抽气阀
15.07 BOOL  ; #4电池抽气阀
15.08 BOOL  ; 13.08
15.09 BOOL  ; #4腔体氦检阀
15.10 BOOL  ; #4腔体破真空阀
15.11 BOOL  ; #4电池破真空阀
15.12 BOOL  ; 吹气电磁阀
15.13 BOOL  ; 扫码NG缓存避位气缸缩回接料
15.14 BOOL  ; 扫码NG缓存接料气缸
15.15 BOOL  ; 扫码NG缓存间隔气缸
1600.00 BOOL  ; SCU21_4 Port#1 Wait Release Switch
1600.01 BOOL  ; SCU21_4 Port#1 Continuous Trace Switch
1600.02 BOOL  ; SCU21_4 Port#1 One-shot Trace Switch
1600.03 BOOL  ; SCU21_4 Port#1 Abort Switch
1600.04 BOOL  ; SCU21_4 Port#1 Serial Gateway Prohibited Switch
1600.05 BOOL  ; SCU21_4 Port#1 Reserved
1600.06 BOOL  ; SCU21_4 Port#1 Loopback Test Switch
1600.07 BOOL  ; SCU21_4 Port#1 Reserved
1600.08 BOOL  ; SCU21_4 Port#2 Wait Release Switch
1600.09 BOOL  ; SCU21_4 Port#2 Continuous Trace Switch
1600.10 BOOL  ; SCU21_4 Port#2 One-shot Trace Switch
1600.11 BOOL  ; SCU21_4 Port#2 Abort Switch
1600.12 BOOL  ; SCU21_4 Port#2 Serial Gateway Prohibited Switch
1600.13 BOOL  ; SCU21_4 Port#2 Reserved
1600.14 BOOL  ; SCU21_4 Port#2 Loopback Test Switch
1600.15 BOOL  ; SCU21_4 Port#2 Reserved
1601.00 BOOL  ; SCU21_4 Protocol Data Error
1601.01 BOOL  ; SCU21_4 Error Log EEPROM Error
1601.02 BOOL  ; SCU21_4 Reserved
1601.03 BOOL  ; SCU21_4 Reserved
1601.04 BOOL  ; SCU21_4 Reserved
1601.05 BOOL  ; SCU21_4 Reserved
1601.06 BOOL  ; SCU21_4 Reserved
1601.07 BOOL  ; SCU21_4 Reserved
1601.08 BOOL  ; SCU21_4 Reserved
1601.09 BOOL  ; SCU21_4 Reserved
1601.10 BOOL  ; SCU21_4 Reserved
1601.11 BOOL  ; SCU21_4 Reserved
1601.12 BOOL  ; SCU21_4 Reserved
1601.13 BOOL  ; SCU21_4 Reserved
1601.14 BOOL  ; SCU21_4 Reserved
1601.15 BOOL  ; SCU21_4 Reserved
1602.00 BOOL  ; SCU21_4 Reserved
1602.01 BOOL  ; SCU21_4 Reserved
1602.02 BOOL  ; SCU21_4 Reserved
1602.03 BOOL  ; SCU21_4 Reserved
1602.04 BOOL  ; SCU21_4 Reserved
1602.05 BOOL  ; SCU21_4 Reserved
1602.06 BOOL  ; SCU21_4 Reserved
1602.07 BOOL  ; SCU21_4 Reserved
1602.08 BOOL  ; SCU21_4 Reserved
1602.09 BOOL  ; SCU21_4 Reserved
1602.10 BOOL  ; SCU21_4 Reserved
1602.11 BOOL  ; SCU21_4 Reserved
1602.12 BOOL  ; SCU21_4 Reserved
1602.13 BOOL  ; SCU21_4 Reserved
1602.14 BOOL  ; SCU21_4 Reserved
1602.15 BOOL  ; SCU21_4 Reserved
1603.00 BOOL  ; SCU21_4 Reserved
1603.01 BOOL  ; SCU21_4 Reserved
1603.02 BOOL  ; SCU21_4 Reserved
1603.03 BOOL  ; SCU21_4 Reserved
1603.04 BOOL  ; SCU21_4 Reserved
1603.05 BOOL  ; SCU21_4 Reserved
1603.06 BOOL  ; SCU21_4 Reserved
1603.07 BOOL  ; SCU21_4 Reserved
1603.08 BOOL  ; SCU21_4 Reserved
1603.09 BOOL  ; SCU21_4 Reserved
1603.10 BOOL  ; SCU21_4 Reserved
1603.11 BOOL  ; SCU21_4 Reserved
1603.12 BOOL  ; SCU21_4 Reserved
1603.13 BOOL  ; SCU21_4 Reserved
1603.14 BOOL  ; SCU21_4 Reserved
1603.15 BOOL  ; SCU21_4 Reserved
1604.00 BOOL  ; SCU21_4 Reserved
1604.01 BOOL  ; SCU21_4 Reserved
1604.02 BOOL  ; SCU21_4 Reserved
1604.03 BOOL  ; SCU21_4 Reserved
1604.04 BOOL  ; SCU21_4 Reserved
1604.05 BOOL  ; SCU21_4 Reserved
1604.06 BOOL  ; SCU21_4 Reserved
1604.07 BOOL  ; SCU21_4 Reserved
1604.08 BOOL  ; SCU21_4 Reserved
1604.09 BOOL  ; SCU21_4 Reserved
1604.10 BOOL  ; SCU21_4 Reserved
1604.11 BOOL  ; SCU21_4 Reserved
1604.12 BOOL  ; SCU21_4 Reserved
1604.13 BOOL  ; SCU21_4 Reserved
1604.14 BOOL  ; SCU21_4 Reserved
1604.15 BOOL  ; SCU21_4 Reserved
1605.00 BOOL  ; SCU21_4 Port#1 Parity: Even/Odd
1605.01 BOOL  ; SCU21_4 Port#1 Parity: Yes/No
1605.02 BOOL  ; SCU21_4 Port#1 Stop bits: 1 or 2 bits
1605.03 BOOL  ; SCU21_4 Port#1 Data length: 7 or 8 bits
1605.04 BOOL  ; SCU21_4 Port#1 Start bits: Always 1
1605.05 BOOL  ; SCU21_4 Port#1 Reserved
1605.06 BOOL  ; SCU21_4 Port#1 Reserved
1605.07 BOOL  ; SCU21_4 Port#1 Reserved
1605.08 BOOL  ; SCU21_4 Port#1 Baud rate
1605.09 BOOL  ; SCU21_4 Port#1 Baud rate
1605.10 BOOL  ; SCU21_4 Port#1 Baud rate
1605.11 BOOL  ; SCU21_4 Port#1 Baud rate
1605.12 BOOL  ; SCU21_4 Port#1 Serial communications mode
1605.13 BOOL  ; SCU21_4 Port#1 Serial communications mode
1605.14 BOOL  ; SCU21_4 Port#1 Serial communications mode
1605.15 BOOL  ; SCU21_4 Port#1 Serial communications mode
1606.00 BOOL  ; SCU21_4 Port#1 1: Port operating; 0: Port stopped
1606.01 BOOL  ; SCU21_4 Port#1 1: System Setup error; 0: System Setup normal
1606.02 BOOL  ; SCU21_4 Port#1 Reserved
1606.03 BOOL  ; SCU21_4 Port#1 Reserved
1606.04 BOOL  ; SCU21_4 Port#1 Reserved
1606.05 BOOL  ; SCU21_4 Port#1 Reserved
1606.06 BOOL  ; SCU21_4 Port#1 Reserved
1606.07 BOOL  ; SCU21_4 Port#1 Reserved
1606.08 BOOL  ; SCU21_4 Port#1 Reserved
1606.09 BOOL  ; SCU21_4 Port#1 Reserved
1606.10 BOOL  ; SCU21_4 Port#1 Reserved
1606.11 BOOL  ; SCU21_4 Port#1 Reserved
1606.12 BOOL  ; SCU21_4 Port#1 Reserved
1606.13 BOOL  ; SCU21_4 Port#1 Terminating resistance
1606.14 BOOL  ; SCU21_4 Port#1 Hardware settings
1606.15 BOOL  ; SCU21_4 Port#1 Hardware settings
1607.00 BOOL  ; SCU21_4 Port#1 Reserved
1607.01 BOOL  ; SCU21_4 Port#1 Reserved
1607.02 BOOL  ; SCU21_4 Port#1 Reserved
1607.03 BOOL  ; SCU21_4 Port#1 RTS (RS) signal
1607.04 BOOL  ; SCU21_4 Port#1 CTS (CS) signal
1607.05 BOOL  ; SCU21_4 Port#1 Reserved
1607.06 BOOL  ; SCU21_4 Port#1 DSR (DR) signal
1607.07 BOOL  ; SCU21_4 Port#1 DTR (ER) signal
1607.08 BOOL  ; SCU21_4 Port#1 Local Unit busy receiving (Flow control)
1607.09 BOOL  ; SCU21_4 Port#1 Reserved
1607.10 BOOL  ; SCU21_4 Port#1 Remote Unit busy receiving (Flow control)
1607.11 BOOL  ; SCU21_4 Port#1 Reserved
1607.12 BOOL  ; SCU21_4 Port#1 Reserved
1607.13 BOOL  ; SCU21_4 Port#1 Reserved
1607.14 BOOL  ; SCU21_4 Port#1 Reserved
1607.15 BOOL  ; SCU21_4 Port#1 Reserved
1608.00 BOOL  ; SCU21_4 Port#1 Reserved
1608.01 BOOL  ; SCU21_4 Port#1 Reserved
1608.02 BOOL  ; SCU21_4 Port#1 Parity error
1608.03 BOOL  ; SCU21_4 Port#1 Framing error
1608.04 BOOL  ; SCU21_4 Port#1 Overrun error
1608.05 BOOL  ; SCU21_4 Port#1 Timeout error
1608.06 BOOL  ; SCU21_4 Port#1 Command error
1608.07 BOOL  ; SCU21_4 Port#1 FCS check error
1608.08 BOOL  ; SCU21_4 Port#1 Number of retries
1608.09 BOOL  ; SCU21_4 Port#1 Number of retries
1608.10 BOOL  ; SCU21_4 Port#1 Number of retries
1608.11 BOOL  ; SCU21_4 Port#1 Number of retries
1608.12 BOOL  ; SCU21_4 Port#1 Tr exceeded
1608.13 BOOL  ; SCU21_4 Port#1 Tfr exceeded
1608.14 BOOL  ; SCU21_4 Port#1 Tfs exceeded
1608.15 BOOL  ; SCU21_4 Port#1 Transmission error
1609.00 BOOL  ; SCU21_4 Port#1 Protocol status
1609.01 BOOL  ; SCU21_4 Port#1 Error codes
1609.02 BOOL  ; SCU21_4 Port#1 Error codes
1609.03 BOOL  ; SCU21_4 Port#1 Error codes
1609.04 BOOL  ; SCU21_4 Port#1 Reserved
1609.05 BOOL  ; SCU21_4 Port#1 Reserved
1609.06 BOOL  ; SCU21_4 Port#1 Reserved
1609.07 BOOL  ; SCU21_4 Port#1 Reserved
1609.08 BOOL  ; SCU21_4 Port#1 Serial Gateway Prohibited Flag
1609.09 BOOL  ; SCU21_4 Port#1 Sequence Waiting Flag
1609.10 BOOL  ; SCU21_4 Port#1 Sequence Abort Completion Flag
1609.11 BOOL  ; SCU21_4 Port#1 Sequence End Completion Flag
1609.12 BOOL  ; SCU21_4 Port#1 Tracing Flag
1609.13 BOOL  ; SCU21_4 Port#1 Aborted Flag
1609.14 BOOL  ; SCU21_4 Port#1 Step Troubleshooting Flag
1610.00 BOOL  ; SCU21_4 Port#1 Communications Sequence Number
1610.01 BOOL  ; SCU21_4 Port#1 Communications Sequence Number
1610.02 BOOL  ; SCU21_4 Port#1 Communications Sequence Number
1610.03 BOOL  ; SCU21_4 Port#1 Communications Sequence Number
1610.04 BOOL  ; SCU21_4 Port#1 Communications Sequence Number
1610.05 BOOL  ; SCU21_4 Port#1 Communications Sequence Number
1610.06 BOOL  ; SCU21_4 Port#1 Communications Sequence Number
1610.07 BOOL  ; SCU21_4 Port#1 Communications Sequence Number
1610.08 BOOL  ; SCU21_4 Port#1 Communications Sequence Number
1610.09 BOOL  ; SCU21_4 Port#1 Communications Sequence Number
1610.10 BOOL  ; SCU21_4 Port#1 Communications Sequence Number
1610.11 BOOL  ; SCU21_4 Port#1 Communications Sequence Number
1610.12 BOOL  ; SCU21_4 Port#1 Reserved
1610.13 BOOL  ; SCU21_4 Port#1 Reserved
1610.14 BOOL  ; SCU21_4 Port#1 Reserved
1610.15 BOOL  ; SCU21_4 Port#1 Reserved
1611.00 BOOL  ; SCU21_4 Port#1 Executed Reception Case Number
1611.01 BOOL  ; SCU21_4 Port#1 Executed Reception Case Number
1611.02 BOOL  ; SCU21_4 Port#1 Executed Reception Case Number
1611.03 BOOL  ; SCU21_4 Port#1 Executed Reception Case Number
1611.04 BOOL  ; SCU21_4 Port#1 Reserved
1611.05 BOOL  ; SCU21_4 Port#1 Reserved
1611.06 BOOL  ; SCU21_4 Port#1 Reserved
1611.07 BOOL  ; SCU21_4 Port#1 Reserved
1611.08 BOOL  ; SCU21_4 Port#1 Executed Step Number
1611.09 BOOL  ; SCU21_4 Port#1 Executed Step Number
1611.10 BOOL  ; SCU21_4 Port#1 Executed Step Number
1611.11 BOOL  ; SCU21_4 Port#1 Executed Step Number
1611.12 BOOL  ; SCU21_4 Port#1 Reserved
1611.13 BOOL  ; SCU21_4 Port#1 Reserved
1611.14 BOOL  ; SCU21_4 Port#1 Reserved
1611.15 BOOL  ; SCU21_4 Port#1 Reserved
1612.00 BOOL  ; SCU21_4 Port#1 Executed Reception Case Number Storage Flag
1612.01 BOOL  ; SCU21_4 Port#1 Executed Reception Case Number Storage Flag
1612.02 BOOL  ; SCU21_4 Port#1 Executed Reception Case Number Storage Flag
1612.03 BOOL  ; SCU21_4 Port#1 Executed Reception Case Number Storage Flag
1612.04 BOOL  ; SCU21_4 Port#1 Executed Reception Case Number Storage Flag
1612.05 BOOL  ; SCU21_4 Port#1 Executed Reception Case Number Storage Flag
1612.06 BOOL  ; SCU21_4 Port#1 Executed Reception Case Number Storage Flag
1612.07 BOOL  ; SCU21_4 Port#1 Executed Reception Case Number Storage Flag
1612.08 BOOL  ; SCU21_4 Port#1 Executed Reception Case Number Storage Flag
1612.09 BOOL  ; SCU21_4 Port#1 Executed Reception Case Number Storage Flag
1612.10 BOOL  ; SCU21_4 Port#1 Executed Reception Case Number Storage Flag
1612.11 BOOL  ; SCU21_4 Port#1 Executed Reception Case Number Storage Flag
1612.12 BOOL  ; SCU21_4 Port#1 Executed Reception Case Number Storage Flag
1612.13 BOOL  ; SCU21_4 Port#1 Executed Reception Case Number Storage Flag
1612.14 BOOL  ; SCU21_4 Port#1 Executed Reception Case Number Storage Flag
1612.15 BOOL  ; SCU21_4 Port#1 Executed Reception Case Number Storage Flag
1613.00 BOOL  ; SCU21_4 Port#1 Executed Step Number Storage Flag
1613.01 BOOL  ; SCU21_4 Port#1 Executed Step Number Storage Flag
1613.02 BOOL  ; SCU21_4 Port#1 Executed Step Number Storage Flag
1613.03 BOOL  ; SCU21_4 Port#1 Executed Step Number Storage Flag
1613.04 BOOL  ; SCU21_4 Port#1 Executed Step Number Storage Flag
1613.05 BOOL  ; SCU21_4 Port#1 Executed Step Number Storage Flag
1613.06 BOOL  ; SCU21_4 Port#1 Executed Step Number Storage Flag
1613.07 BOOL  ; SCU21_4 Port#1 Executed Step Number Storage Flag
1613.08 BOOL  ; SCU21_4 Port#1 Executed Step Number Storage Flag
1613.09 BOOL  ; SCU21_4 Port#1 Executed Step Number Storage Flag
1613.10 BOOL  ; SCU21_4 Port#1 Executed Step Number Storage Flag
1613.11 BOOL  ; SCU21_4 Port#1 Executed Step Number Storage Flag
1613.12 BOOL  ; SCU21_4 Port#1 Executed Step Number Storage Flag
1613.13 BOOL  ; SCU21_4 Port#1 Executed Step Number Storage Flag
1613.14 BOOL  ; SCU21_4 Port#1 Executed Step Number Storage Flag
1613.15 BOOL  ; SCU21_4 Port#1 Executed Step Number Storage Flag
1614.00 BOOL  ; SCU21_4 Port#1 Repeat Counter Present Value
1614.01 BOOL  ; SCU21_4 Port#1 Repeat Counter Present Value
1614.02 BOOL  ; SCU21_4 Port#1 Repeat Counter Present Value
1614.03 BOOL  ; SCU21_4 Port#1 Repeat Counter Present Value
1614.04 BOOL  ; SCU21_4 Port#1 Repeat Counter Present Value
1614.05 BOOL  ; SCU21_4 Port#1 Repeat Counter Present Value
1614.06 BOOL  ; SCU21_4 Port#1 Repeat Counter Present Value
1614.07 BOOL  ; SCU21_4 Port#1 Repeat Counter Present Value
1614.08 BOOL  ; SCU21_4 Port#1 Repeat Counter Setting Value
1614.09 BOOL  ; SCU21_4 Port#1 Repeat Counter Setting Value
1614.10 BOOL  ; SCU21_4 Port#1 Repeat Counter Setting Value
1614.11 BOOL  ; SCU21_4 Port#1 Repeat Counter Setting Value
1614.12 BOOL  ; SCU21_4 Port#1 Repeat Counter Setting Value
1614.13 BOOL  ; SCU21_4 Port#1 Repeat Counter Setting Value
1614.14 BOOL  ; SCU21_4 Port#1 Repeat Counter Setting Value
1614.15 BOOL  ; SCU21_4 Port#1 Repeat Counter Setting Value
1615.00 BOOL  ; SCU21_4 Port#2 Parity: Even/Odd
1615.01 BOOL  ; SCU21_4 Port#2 Parity: Yes/No
1615.02 BOOL  ; SCU21_4 Port#2 Stop bits: 1 or 2 bits
1615.03 BOOL  ; SCU21_4 Port#2 Data length: 7 or 8 bits
1615.04 BOOL  ; SCU21_4 Port#2 Start bits: Always 1
1615.05 BOOL  ; SCU21_4 Port#2 Reserved
1615.06 BOOL  ; SCU21_4 Port#2 Reserved
1615.07 BOOL  ; SCU21_4 Port#2 Reserved
1615.08 BOOL  ; SCU21_4 Port#2 Baud rate
1615.09 BOOL  ; SCU21_4 Port#2 Baud rate
1615.10 BOOL  ; SCU21_4 Port#2 Baud rate
1615.11 BOOL  ; SCU21_4 Port#2 Baud rate
1615.12 BOOL  ; SCU21_4 Port#2 Serial communications mode
1615.13 BOOL  ; SCU21_4 Port#2 Serial communications mode
1615.14 BOOL  ; SCU21_4 Port#2 Serial communications mode
1615.15 BOOL  ; SCU21_4 Port#2 Serial communications mode
1616.00 BOOL  ; SCU21_4 Port#2 1: Port operating; 0: Port stopped
1616.01 BOOL  ; SCU21_4 Port#2 1: System Setup error; 0: System Setup normal
1616.02 BOOL  ; SCU21_4 Port#2 Reserved
1616.03 BOOL  ; SCU21_4 Port#2 Reserved
1616.04 BOOL  ; SCU21_4 Port#2 Reserved
1616.05 BOOL  ; SCU21_4 Port#2 Reserved
1616.06 BOOL  ; SCU21_4 Port#2 Reserved
1616.07 BOOL  ; SCU21_4 Port#2 Reserved
1616.08 BOOL  ; SCU21_4 Port#2 Reserved
1616.09 BOOL  ; SCU21_4 Port#2 Reserved
1616.10 BOOL  ; SCU21_4 Port#2 Reserved
1616.11 BOOL  ; SCU21_4 Port#2 Reserved
1616.12 BOOL  ; SCU21_4 Port#2 Reserved
1616.13 BOOL  ; SCU21_4 Port#2 Terminating resistance
1616.14 BOOL  ; SCU21_4 Port#2 Hardware settings
1616.15 BOOL  ; SCU21_4 Port#2 Hardware settings
1617.00 BOOL  ; SCU21_4 Port#2 Reserved
1617.01 BOOL  ; SCU21_4 Port#2 Reserved
1617.02 BOOL  ; SCU21_4 Port#2 Reserved
1617.03 BOOL  ; SCU21_4 Port#2 RTS (RS) signal
1617.04 BOOL  ; SCU21_4 Port#2 CTS (CS) signal
1617.05 BOOL  ; SCU21_4 Port#2 Reserved
1617.06 BOOL  ; SCU21_4 Port#2 DSR (DR) signal
1617.07 BOOL  ; SCU21_4 Port#2 DTR (ER) signal
1617.08 BOOL  ; SCU21_4 Port#2 Local Unit busy receiving (Flow control)
1617.09 BOOL  ; SCU21_4 Port#2 Reserved
1617.10 BOOL  ; SCU21_4 Port#2 Remote Unit busy receiving (Flow control)
1617.11 BOOL  ; SCU21_4 Port#2 Reserved
1617.12 BOOL  ; SCU21_4 Port#2 Reserved
1617.13 BOOL  ; SCU21_4 Port#2 Reserved
1617.14 BOOL  ; SCU21_4 Port#2 Reserved
1617.15 BOOL  ; SCU21_4 Port#2 Reserved
1618.00 BOOL  ; SCU21_4 Port#2 Reserved
1618.01 BOOL  ; SCU21_4 Port#2 Reserved
1618.02 BOOL  ; SCU21_4 Port#2 Parity error
1618.03 BOOL  ; SCU21_4 Port#2 Framing error
1618.04 BOOL  ; SCU21_4 Port#2 Overrun error
1618.05 BOOL  ; SCU21_4 Port#2 Timeout error
1618.06 BOOL  ; SCU21_4 Port#2 Command error
1618.07 BOOL  ; SCU21_4 Port#2 FCS check error
1618.08 BOOL  ; SCU21_4 Port#2 Number of retries
1618.09 BOOL  ; SCU21_4 Port#2 Number of retries
1618.10 BOOL  ; SCU21_4 Port#2 Number of retries
1618.11 BOOL  ; SCU21_4 Port#2 Number of retries
1618.12 BOOL  ; SCU21_4 Port#2 Tr exceeded
1618.13 BOOL  ; SCU21_4 Port#2 Tfr exceeded
1618.14 BOOL  ; SCU21_4 Port#2 Tfs exceeded
1618.15 BOOL  ; SCU21_4 Port#2 Transmission error
1619.00 BOOL  ; SCU21_4 Port#2 Protocol status
1619.01 BOOL  ; SCU21_4 Port#2 Error codes
1619.02 BOOL  ; SCU21_4 Port#2 Error codes
1619.03 BOOL  ; SCU21_4 Port#2 Error codes
1619.04 BOOL  ; SCU21_4 Port#2 Reserved
1619.05 BOOL  ; SCU21_4 Port#2 Reserved
1619.06 BOOL  ; SCU21_4 Port#2 Reserved
1619.07 BOOL  ; SCU21_4 Port#2 Reserved
1619.08 BOOL  ; SCU21_4 Port#2 Serial Gateway Prohibited Flag
1619.09 BOOL  ; SCU21_4 Port#2 Sequence Waiting Flag
1619.10 BOOL  ; SCU21_4 Port#2 Sequence Abort Completion Flag
1619.11 BOOL  ; SCU21_4 Port#2 Sequence End Completion Flag
1619.12 BOOL  ; SCU21_4 Port#2 Tracing Flag
1619.13 BOOL  ; SCU21_4 Port#2 Aborted Flag
1619.14 BOOL  ; SCU21_4 Port#2 Step Troubleshooting Flag
1619.15 BOOL  ; SCU21_4 Port#2 Protocol Macro Executing Flag
1620.00 BOOL  ; SCU21_4 Port#2 Communications Sequence Number
1620.01 BOOL  ; SCU21_4 Port#2 Communications Sequence Number
1620.02 BOOL  ; SCU21_4 Port#2 Communications Sequence Number
1620.03 BOOL  ; SCU21_4 Port#2 Communications Sequence Number
1620.04 BOOL  ; SCU21_4 Port#2 Communications Sequence Number
1620.05 BOOL  ; SCU21_4 Port#2 Communications Sequence Number
1620.06 BOOL  ; SCU21_4 Port#2 Communications Sequence Number
1620.07 BOOL  ; SCU21_4 Port#2 Communications Sequence Number
1620.08 BOOL  ; SCU21_4 Port#2 Communications Sequence Number
1620.09 BOOL  ; SCU21_4 Port#2 Communications Sequence Number
1620.10 BOOL  ; SCU21_4 Port#2 Communications Sequence Number
1620.11 BOOL  ; SCU21_4 Port#2 Communications Sequence Number
1620.12 BOOL  ; SCU21_4 Port#2 Reserved
1620.13 BOOL  ; SCU21_4 Port#2 Reserved
1620.14 BOOL  ; SCU21_4 Port#2 Reserved
1620.15 BOOL  ; SCU21_4 Port#2 Reserved
1621.00 BOOL  ; SCU21_4 Port#2 Executed Reception Case Number
1621.01 BOOL  ; SCU21_4 Port#2 Executed Reception Case Number
1621.02 BOOL  ; SCU21_4 Port#2 Executed Reception Case Number
1621.03 BOOL  ; SCU21_4 Port#2 Executed Reception Case Number
1621.04 BOOL  ; SCU21_4 Port#2 Reserved
1621.05 BOOL  ; SCU21_4 Port#2 Reserved
1621.06 BOOL  ; SCU21_4 Port#2 Reserved
1621.07 BOOL  ; SCU21_4 Port#2 Reserved
1621.08 BOOL  ; SCU21_4 Port#2 Executed Step Number
1621.09 BOOL  ; SCU21_4 Port#2 Executed Step Number
1621.10 BOOL  ; SCU21_4 Port#2 Executed Step Number
1621.11 BOOL  ; SCU21_4 Port#2 Executed Step Number
1621.12 BOOL  ; SCU21_4 Port#2 Reserved
1621.13 BOOL  ; SCU21_4 Port#2 Reserved
1621.14 BOOL  ; SCU21_4 Port#2 Reserved
1621.15 BOOL  ; SCU21_4 Port#2 Reserved
1622.00 BOOL  ; SCU21_4 Port#2 Executed Reception Case Number Storage Flag
1622.01 BOOL  ; SCU21_4 Port#2 Executed Reception Case Number Storage Flag
1622.02 BOOL  ; SCU21_4 Port#2 Executed Reception Case Number Storage Flag
1622.03 BOOL  ; SCU21_4 Port#2 Executed Reception Case Number Storage Flag
1622.04 BOOL  ; SCU21_4 Port#2 Executed Reception Case Number Storage Flag
1622.05 BOOL  ; SCU21_4 Port#2 Executed Reception Case Number Storage Flag
1622.06 BOOL  ; SCU21_4 Port#2 Executed Reception Case Number Storage Flag
1622.07 BOOL  ; SCU21_4 Port#2 Executed Reception Case Number Storage Flag
1622.08 BOOL  ; SCU21_4 Port#2 Executed Reception Case Number Storage Flag
1622.09 BOOL  ; SCU21_4 Port#2 Executed Reception Case Number Storage Flag
1622.10 BOOL  ; SCU21_4 Port#2 Executed Reception Case Number Storage Flag
1622.11 BOOL  ; SCU21_4 Port#2 Executed Reception Case Number Storage Flag
1622.12 BOOL  ; SCU21_4 Port#2 Executed Reception Case Number Storage Flag
1622.13 BOOL  ; SCU21_4 Port#2 Executed Reception Case Number Storage Flag
1622.14 BOOL  ; SCU21_4 Port#2 Executed Reception Case Number Storage Flag
1622.15 BOOL  ; SCU21_4 Port#2 Executed Reception Case Number Storage Flag
1623.00 BOOL  ; SCU21_4 Port#2 Executed Step Number Storage Flag
1623.01 BOOL  ; SCU21_4 Port#2 Executed Step Number Storage Flag
1623.02 BOOL  ; SCU21_4 Port#2 Executed Step Number Storage Flag
1623.03 BOOL  ; SCU21_4 Port#2 Executed Step Number Storage Flag
1623.04 BOOL  ; SCU21_4 Port#2 Executed Step Number Storage Flag
1623.05 BOOL  ; SCU21_4 Port#2 Executed Step Number Storage Flag
1623.06 BOOL  ; SCU21_4 Port#2 Executed Step Number Storage Flag
1623.07 BOOL  ; SCU21_4 Port#2 Executed Step Number Storage Flag
1623.08 BOOL  ; SCU21_4 Port#2 Executed Step Number Storage Flag
1623.09 BOOL  ; SCU21_4 Port#2 Executed Step Number Storage Flag
1623.10 BOOL  ; SCU21_4 Port#2 Executed Step Number Storage Flag
1623.11 BOOL  ; SCU21_4 Port#2 Executed Step Number Storage Flag
1623.12 BOOL  ; SCU21_4 Port#2 Executed Step Number Storage Flag
1623.13 BOOL  ; SCU21_4 Port#2 Executed Step Number Storage Flag
1623.14 BOOL  ; SCU21_4 Port#2 Executed Step Number Storage Flag
1623.15 BOOL  ; SCU21_4 Port#2 Executed Step Number Storage Flag
1624.00 BOOL  ; SCU21_4 Port#2 Repeat Counter Present Value
1624.01 BOOL  ; SCU21_4 Port#2 Repeat Counter Present Value
1624.02 BOOL  ; SCU21_4 Port#2 Repeat Counter Present Value
1624.03 BOOL  ; SCU21_4 Port#2 Repeat Counter Present Value
1624.04 BOOL  ; SCU21_4 Port#2 Repeat Counter Present Value
1624.05 BOOL  ; SCU21_4 Port#2 Repeat Counter Present Value
1624.06 BOOL  ; SCU21_4 Port#2 Repeat Counter Present Value
1624.07 BOOL  ; SCU21_4 Port#2 Repeat Counter Present Value
1624.08 BOOL  ; SCU21_4 Port#2 Repeat Counter Setting Value
1624.09 BOOL  ; SCU21_4 Port#2 Repeat Counter Setting Value
1624.10 BOOL  ; SCU21_4 Port#2 Repeat Counter Setting Value
1624.11 BOOL  ; SCU21_4 Port#2 Repeat Counter Setting Value
1624.12 BOOL  ; SCU21_4 Port#2 Repeat Counter Setting Value
1624.13 BOOL  ; SCU21_4 Port#2 Repeat Counter Setting Value
1624.14 BOOL  ; SCU21_4 Port#2 Repeat Counter Setting Value
1624.15 BOOL  ; SCU21_4 Port#2 Repeat Counter Setting Value
162.00 BOOL  ; 进料升降伺服归零(M)
162.01 BOOL  ; 进料升降伺服点动下降(M)
162.02 BOOL  ; 进料升降伺服点动上升
162.03 BOOL  ; 进料升降伺服到取料位
162.04 BOOL  ; 进料升降伺服到放料位
162.09 BOOL  ; 进料升降伺服手动运转条件
162.11 BOOL  ; 进料升降伺服手动定位条件
162.12 BOOL  ; 进料升降伺服手动定位(M)
162.13 BOOL  ; 进料升降伺服手动定位
164.00 BOOL  ; 升降伺服下降取料
164.01 BOOL  ; 升降伺服上回零
164.02 BOOL  ; 升降伺服放料下降
164.03 BOOL  ; 进料升降伺放料后上升
164.09 BOOL  ; 进料升降伺服归零(复位)(M)
173.00 BOOL  ; 出料升降伺服归零
173.01 BOOL  ; 出料升降伺服点动下降(M)
173.02 BOOL  ; 出料升伺服点动上升
173.03 BOOL  ; nc
173.04 BOOL  ; 出料升降伺服到取料高度
173.05 BOOL  ; 出料升降伺服到放料高度(M)
173.09 BOOL  ; 出料升降伺服回原条件
173.10 BOOL  ; 出料升降伺服复位
173.11 BOOL  ; 出料升降伺服手动定位条件
173.12 BOOL  ; 出料升降伺服手动定位(M)
173.13 BOOL  ; 出料升降伺服手动定位
174.00 BOOL  ; 出料升降下取料
174.01 BOOL  ; 出料升降伺服回零
174.02 BOOL  ; 下降放料
174.03 BOOL  ; 放料上升
180.01 BOOL  ; #1腔体抽气阀
180.02 BOOL  ; #2腔体抽气阀
180.03 BOOL  ; #3腔体抽气阀
180.04 BOOL  ; #4腔体抽气阀
190.00 BOOL  ; #1腔体抽残气时停止
190.01 BOOL  ; #2腔体抽残气时停止
190.02 BOOL  ; #3腔体抽残气时停止
190.03 BOOL  ; #4腔体抽残气时停止
19.00 BOOL  ; 没有氦检阀打开
1.00 BOOL  ; 测试NG#1托盘有料
1.01 BOOL  ; 测试NG#2托盘有料
1.02 BOOL  ; 测试NG#3托盘有料
1.03 BOOL  ; 测试NG#4托盘有料
1.04 BOOL  ; 上料夹爪柔性报警
1.05 BOOL  ; 下料夹爪柔性报警
1.06 BOOL  ; 前腔体进料柔性报警
1.07 BOOL  ; 后腔体进料柔性报警
1.08 BOOL  ; 前腔体出料柔性报警
1.09 BOOL  ; 后腔体出料柔性报警
1.10 BOOL  ; #1真空泵缺相
1.11 BOOL  ; #2真空泵缺相
1.12 BOOL  ; 氦检仪异常
1.13 BOOL  ; 总气源开关
1.14 BOOL  ; 启动按钮
1.15 BOOL  ; 停止按钮
2000.00 BOOL  ; 进料伺服序列号使能
2000.01 BOOL  ; 进料伺服起动
2000.02 BOOL  ; 进料伺服独立起动
2000.03 BOOL  ; 进料水平移载伺服绝对移动
2000.04 BOOL  ; 进料伺服相对移动
2000.05 BOOL  ; 进料伺服中断进给
2000.06 BOOL  ; 进料伺服原点搜索
2000.07 BOOL  ; 进料伺服原点返回
2000.08 BOOL  ; 进料伺服当前位置预置
2000.09 BOOL  ; 进料水平移载伺服点动
2000.10 BOOL  ; 进料水平移载伺服方向定义
2000.11 BOOL  ; 进料伺服示教
2000.12 BOOL  ; 进料水平移载伺服释放禁止/复位
2000.13 BOOL  ; 进料伺服偏差计数器复位输出/原点调整命令输出
2000.14 BOOL  ; 进料伺服激活Override
2000.15 BOOL  ; 进料伺服停止
2001.08 BOOL  ; 进料伺服强迫中断
2001.12 BOOL  ; 进料伺服写数据
2001.13 BOOL  ; 进料伺服读数据
2001.14 BOOL  ; 进料伺服保存数据
2002.00 BOOL  ; 出料伺服序列号使能
2002.01 BOOL  ; 出料伺服起动
2002.02 BOOL  ; 出料伺服独立起动
2002.03 BOOL  ; 出料伺服绝对移动
2002.04 BOOL  ; 出料伺服相对移动
2002.05 BOOL  ; 出料伺服中断进给
2002.06 BOOL  ; 出料水平移载伺服原点搜索
2002.07 BOOL  ; 出料伺服原点返回
2002.08 BOOL  ; 出料伺服当前位置预置
2002.09 BOOL  ; 出料伺服点动
2002.10 BOOL  ; 出料伺服方向定义
2002.11 BOOL  ; 出料伺服示教
2002.12 BOOL  ; 出料伺服释放禁止/复位
2002.13 BOOL  ; 出料伺服偏差计数器复位输出/原点调整命令输出
2002.14 BOOL  ; 出料伺服激活Override
2002.15 BOOL  ; 出料伺服停止
2003.08 BOOL  ; 出料伺服强迫中断
2003.12 BOOL  ; 出料伺服写数据
2003.13 BOOL  ; 出料伺服读数据
2003.14 BOOL  ; 出料伺服保存数据
2004.03 BOOL  ; 进料升降伺服绝对移动
2004.04 BOOL  ; 进料伺服等待存储器操作标志位
2004.05 BOOL  ; 进料伺服定位结束标志位
2004.06 BOOL  ; 进料升降伺服原点搜索
2004.08 BOOL  ; 进料伺服区域0监控标志位
2004.09 BOOL  ; 进料升降伺服点动
2004.10 BOOL  ; 进料升降伺服方向定义
2004.11 BOOL  ; 进料伺服示教完成标志位
2004.12 BOOL  ; 进料升降伺服释放禁止/复位
2004.14 BOOL  ; 进料伺服数据传送标志
2004.15 BOOL  ; 进料伺服减速停止执行标志
2005.10 BOOL  ; 进料伺服原点接近输入信号
2005.11 BOOL  ; 进料伺服原点输入信号
2005.12 BOOL  ; 进料伺服中断输入信号
2005.13 BOOL  ; 进料伺服紧急停止输入信号
2005.14 BOOL  ; 进料伺服定位完成信号
2005.15 BOOL  ; 进料伺服偏差计数器复位输出/原点调整命令输出
2006.03 BOOL  ; 出料升降伺服绝对移动
2006.06 BOOL  ; 出料升降伺服原点搜索
2006.09 BOOL  ; 出料升降伺服点动
2006.10 BOOL  ; 出料升降伺服方向定义
2006.12 BOOL  ; 出料伺服报警复位
2007.04 BOOL  ; 出料伺服等待存储器操作标志位
2007.05 BOOL  ; 出料伺服定位结束标志位
2007.08 BOOL  ; 出料伺服区域0监控标志位
2007.09 BOOL  ; 出料伺服区域1监控标志位
2007.10 BOOL  ; 出料伺服区域2监控标志位
2007.11 BOOL  ; 出料伺服示教完成标志位
2007.12 BOOL  ; 出料伺服标志位
2007.14 BOOL  ; 出料伺服数据传送标志
2007.15 BOOL  ; 出料伺服减速停止执行标志
2008.06 BOOL  ; 进料伺服无原点标志位
2008.07 BOOL  ; 进料伺服原点停止标志位
2008.10 BOOL  ; 出料伺服原点接近输入信号
2008.11 BOOL  ; 出料伺服原点输入信号
2008.12 BOOL  ; 出料伺服中断输入信号
2008.13 BOOL  ; 进料移载伺服忙标志位
2008.14 BOOL  ; 出料伺服定位完成信号
2008.15 BOOL  ; 出料伺服偏差计数器复位输出/原点调整命令输出
2009.08 BOOL  ; 进料伺服前极限输入信号
2009.09 BOOL  ; 进料伺服后极限输入信号
2010 CHANNEL  ; 进料伺服错误代码
2011.06 BOOL  ; 出料伺服无原点标志位
2011.07 BOOL  ; 出料伺服原点停止标志位
2011.13 BOOL  ; 出料移载伺服忙标志位
2012.08 BOOL  ; 出料伺服CW极限输入信号
2012.09 BOOL  ; 出料伺服CCW极限输入信号
2013 CHANNEL  ; 出料伺服错误代码
2014.06 BOOL  ; 进料升降伺服无原点标志位
2014.13 BOOL  ; 进料升降伺服忙标志位
2015.08 BOOL  ; 进料升降伺服下极限输入信号
2015.09 BOOL  ; 进料升降伺服上极限输入信号
2015.11 BOOL  ; 进料升降伺服原点
2017.06 BOOL  ; 出料升降伺服无原点标志位
2017.13 BOOL  ; 出料升降伺服忙标志位
2018.08 BOOL  ; 出料升降伺服CW极限输入信号
2018.09 BOOL  ; 出料升降伺服CCW极限输入信号
2018.11 BOOL  ; 出料升降伺服原点
2018.13 BOOL  ; 出料升降伺服忙标志位
2021 CHANNEL  ; 1#腔体真空计模拟量读数(AD041_1)
2022 CHANNEL  ; 2#腔体真空计模拟量读数(AD041_2)
2023 CHANNEL  ; 3#腔体真空计模拟量读数(AD041_3)
2024 CHANNEL  ; 4#腔体真空计模拟量读数(AD041_4)
2025 CHANNEL  ; 5#模拟量读数(AD081_5)
2026 CHANNEL  ; 6#模拟量读数(AD081_6)
2027 CHANNEL  ; 7#模拟量读数(AD081_7)
2028 CHANNEL  ; 8#模拟量读数(AD081_8)
2029 CHANNEL  ; AD081错误代码
2029.00 BOOL  ; 1#真空计断线
2029.01 BOOL  ; 2#真空计断线
2029.02 BOOL  ; 3#真空计断线
2029.03 BOOL  ; 4#真空计断线
2029.04 BOOL  ; 1#密封气缸压力表断线
2029.05 BOOL  ; 2#密封气缸压力表断线
2029.06 BOOL  ; 3#密封气缸压力表断线
2029.07 BOOL  ; 4#密封气缸压力表断线
20.00 BOOL  ; 自动模式切换按钮(T)
20.01 BOOL  ; 自动启动按钮(T)
20.02 BOOL  ; 自动停止按钮(T)
20.03 BOOL  ; 清料停止按钮(T)
20.04 BOOL  ; 蜂鸣器停止按钮(T)
20.05 BOOL  ; 错误清除按钮(T)
20.06 BOOL  ; 出料拉带记忆清除按钮(T)
20.07 BOOL  ; 柔性报警解除按钮(T)
20.08 BOOL  ; 电池测试NG报警解除按钮(T)
20.09 BOOL  ; 缓存满料报警解除(T)
20.10 BOOL  ; 重新扫码按钮(T)(A)
20.11 BOOL  ; MES校验错误确认按钮(T)
20.12 BOOL  ; MES模式打开按钮
20.13 BOOL  ; MES弹出窗口取消按钮
20.14 BOOL  ; 清氦失败后再次清氦按钮
20.15 BOOL  ; 清氦失败后跳过再次清氦按钮
21.00 BOOL  ; 整机复位按钮(T)
21.01 BOOL  ; 整机记忆清除按钮(T)
21.02 BOOL  ; 生产总数清零按钮(T)
21.03 BOOL  ; 生产OK数清零按钮(T)
21.04 BOOL  ; 生产NG数清零按钮(T)
21.10 BOOL  ; 伺服参数确认按钮(T)
21.11 BOOL  ; 进料MES校验NG电池已取走确认按钮(T)
22.00 BOOL  ; 寸动模式
230.00 BOOL  ; 前腔体进料顶升伸出
230.01 BOOL  ; 前腔体进料顶升缩回
230.02 BOOL  ; 进料#2升降气缸上升(M)
230.03 BOOL  ; 进料#2升降气缸下降(M)
230.04 BOOL  ; 后腔体进料顶升伸出
230.05 BOOL  ; 后腔体进料顶升缩回
23.00 BOOL  ; 进料机构记忆清除
23.01 BOOL  ; 前进料缓存记忆清除
23.02 BOOL  ; 后进料缓存记忆清除
23.03 BOOL  ; 前上料记忆清除
23.04 BOOL  ; 前下料记忆清除
23.05 BOOL  ; 后上料记忆清除
23.06 BOOL  ; 后下料记忆清除
23.07 BOOL  ; #1腔体记忆清除
23.08 BOOL  ; #2腔体记忆清除
23.09 BOOL  ; #3腔体记忆清除
23.10 BOOL  ; #4腔体记忆清除
23.11 BOOL  ; 出料夹爪记忆清除
23.12 BOOL  ; 前出料缓存记忆清除
23.13 BOOL  ; 后出料缓存记忆清除
23.14 BOOL  ; 拉带上料位记忆清除
241.04 BOOL  ; 出料#2升降气缸上升(M)
241.05 BOOL  ; 出料#1升降气缸下降(M)
243.00 BOOL  ; 出料伺服回原条件
26 CHANNEL  ; 氦检仪数值稳定延时
2960.00 BOOL  ; 前腔体上料伺服原点
2960.01 BOOL  ; 前腔体上料伺服原点接近
2960.02 BOOL  ; 前腔体取料伺服原点
2960.03 BOOL  ; 前腔体取料伺服原点接近
2960.06 BOOL  ; 前腔体上料伺服反转极限
2960.07 BOOL  ; 前腔体上料伺服正转极限
2960.08 BOOL  ; 前腔体取料伺服反转极限
2960.09 BOOL  ; 前腔体取料伺服正转极限
2961.00 BOOL  ; 前腔体上料伺服脉冲
2961.01 BOOL  ; 前腔体取料伺服脉冲
2961.02 BOOL  ; 前腔体上料伺服方向
2961.03 BOOL  ; 前腔体取料伺服方向
2962.00 BOOL  ; 后腔体上料伺服原点
2962.01 BOOL  ; 后腔体上料伺服原点接近
2962.02 BOOL  ; 后腔体取料伺服原点
2962.03 BOOL  ; 后腔体取料伺服原点接近
2962.06 BOOL  ; 后腔体上料伺服正转极限
2962.07 BOOL  ; 后腔体上料伺服反转极限
2962.08 BOOL  ; 后腔体取料伺服正转极限
2962.09 BOOL  ; 后腔体取料伺服反转极限
2963.00 BOOL  ; 后腔体上料伺服脉冲
2963.01 BOOL  ; 后腔体取料伺服脉冲
2963.02 BOOL  ; 后腔体上料伺服方向
2963.03 BOOL  ; 后腔体取料伺服方向
2963.04 BOOL  ; 后上料伺服原点回归完成标志
2963.05 BOOL  ; 后下料伺服原点回归完成标志
2.00 BOOL  ; 复位按钮
2.01 BOOL  ; 急停按钮
2.02 BOOL  ; 前门磁开关
2.03 BOOL  ; 后门磁开关
2.04 BOOL  ; 左门磁开关
2.05 BOOL  ; 右门磁开关
2.06 BOOL  ; 进料移栽伺服Ready
2.07 BOOL  ; 进料移栽伺服Alarm
2.08 BOOL  ; 出料移栽伺服Ready
2.09 BOOL  ; 出料移栽伺服Alarm
2.10 BOOL  ; 前腔体进料伺服Ready
2.11 BOOL  ; 前腔体进料伺服Alarm
2.12 BOOL  ; 后腔体进料伺服Ready
2.13 BOOL  ; 后腔体进料伺服Alarm
2.14 BOOL  ; 前腔体出料伺服Ready
2.15 BOOL  ; 前腔体出料伺服Alarm
300.06 BOOL  ; debug
30.00 BOOL  ; 扫码阻挡气缸-HMI
30.01 BOOL  ; 上料#1升降气缸-HMI
30.02 BOOL  ; 上料#2级升降M
30.03 BOOL  ; 扫码气缸下降按钮(T)
30.04 BOOL  ; 进料升降气缸上升按钮(T)
30.05 BOOL  ; #1扫码NG气缸按钮(T)
30.06 BOOL  ; #2扫码NG气缸按钮(T)
30.07 BOOL  ; 进料平移气缸合按钮(T)
30.08 BOOL  ; 进料顶升气缸张开按钮(T)
30.09 BOOL  ; 夹紧阻挡气缸按钮(T)
30.10 BOOL  ; 进料电机手动
30.11 BOOL  ; 下料横移气缸按钮(T)
30.12 BOOL  ; 后进料旋转气缸转回按钮(T)
30.13 BOOL  ; 后进料旋转气缸旋转按钮(T)
30.14 BOOL  ; 避位气缸接料按钮(T)
30.15 BOOL  ; 避位气缸避位伸出按钮(T)
31.00 BOOL  ; 接料气缸前进按钮(T)
31.01 BOOL  ; 接料气缸后退按钮(T)
31.02 BOOL  ; 间隔气缸上升按钮(T)
31.03 BOOL  ; 间隔气缸下降按钮(T)
31.05 BOOL  ; 右扫码按钮(T)
31.06 BOOL  ; 放弃扫码-hmi
31.08 BOOL  ; 进料夹子松开-HMI
31.10 BOOL  ; 进料#1扫码NG位置按钮
31.11 BOOL  ; 进料#2扫码NG位置按钮
31.12 BOOL  ; 进料伺服到#3扫码NG位
31.13 BOOL  ; 进料伺服到#4扫码NG位
32.00 BOOL  ; 进料伺服归零按钮(T)
32.01 BOOL  ; 进料伺服点动前进按钮(T)
32.02 BOOL  ; 进料伺服点动后退按钮(T)
32.03 BOOL  ; 进料#4扫码NG位置按钮(T)
32.04 BOOL  ; 进料伺服到取料位置按钮(T)
32.05 BOOL  ; 进料伺服到前放料位置按钮(T)
32.06 BOOL  ; 进料伺服到后放料位置按钮(T)
32.07 BOOL  ; 进料#2扫码NG位设定按钮(T)
32.08 BOOL  ; 进料#3扫码NG位设定按钮(T)
32.09 BOOL  ; 进料#4扫码NG位设定按钮(T)
32.10 BOOL  ; 进料伺服取料位设定按钮(T)
32.11 BOOL  ; 进料伺服前放料位设定按钮(T)
32.12 BOOL  ; 进料伺服后放料位设定按钮(T)
32.13 BOOL  ; 进料#1扫码NG位设定按钮(T)
32.14 BOOL  ; 进料机构单次循环按钮(T)
32.15 BOOL  ; 进料机构复位按钮(T)
33.00 BOOL  ; 前上料升降气缸下降按钮
33.01 BOOL  ; 前上料夹爪气缸松开按钮
33.02 BOOL  ; 前上料2级升降气缸上升按钮
33.03 BOOL  ; 前上料2级升降气缸下降按钮
33.04 BOOL  ; 前上料夹爪气缸夹紧按钮
33.05 BOOL  ; 前上料夹爪气缸松开按钮
34.00 BOOL  ; 前上料伺服归零按钮(T)
34.01 BOOL  ; 前上料伺服点动前进按钮(T)
34.02 BOOL  ; 前上料伺服点动后退按钮(T)
34.03 BOOL  ; 前上料伺服到等待位置按钮(T)
34.04 BOOL  ; 前上料伺服到取料位置按钮(T)
34.05 BOOL  ; 前上料伺服到仓1放料位置按钮(T)
34.06 BOOL  ; 前上料伺服到仓2放料位置按钮(T)
34.09 BOOL  ; 前上料伺服等待位设定按钮(T)
34.10 BOOL  ; 前上料伺服取料位设定按钮(T)
34.11 BOOL  ; 前上料伺服仓1放料位设定按钮(T)
34.12 BOOL  ; 前上料伺服仓2放料位设定按钮(T)
34.14 BOOL  ; 前上料机构单次循环按钮(T)
34.15 BOOL  ; 前上料机构复位按钮(T)
35.00 BOOL  ; 前下料升降气缸下降按钮
35.01 BOOL  ; 前下料夹爪气缸松开按钮
35.02 BOOL  ; 前下料2级升降气缸上升按钮
35.03 BOOL  ; 前下料2级升降气缸下降按钮
35.04 BOOL  ; 前下料夹爪气缸夹紧按钮
35.05 BOOL  ; 前下料夹爪气缸松开按钮
35.10 BOOL  ; 腔体1检测开始位
35.11 BOOL  ; 腔体1检测结束位
35.12 BOOL  ; 腔体2检测开始位
35.13 BOOL  ; 腔体2检测结束位
36.00 BOOL  ; 前下料伺服归零按钮(T)
36.01 BOOL  ; 前下料伺服点动前进按钮(T)
36.02 BOOL  ; 前下料伺服点动后退按钮(T)
36.03 BOOL  ; 前下料伺服到等待位置按钮(T)
36.04 BOOL  ; 前下料伺服到仓1取料位置按钮(T)
36.05 BOOL  ; 前下料伺服到仓2取料位置按钮(T)
36.06 BOOL  ; 前下料伺服到放料位置按钮(T)
36.07 BOOL  ; 前下料伺服到NG放料位置按钮(T)
36.09 BOOL  ; 前下料伺服等待位设定按钮(T)
36.10 BOOL  ; 前下料伺服仓1取料位设定按钮(T)
36.11 BOOL  ; 前下料伺服仓2取料位设定按钮(T)
36.12 BOOL  ; 前下料伺服放料位设定按钮(T)
36.13 BOOL  ; 前下料伺服NG放料位设定按钮(T)
36.14 BOOL  ; 前下料机构单次循环按钮(T)
36.15 BOOL  ; 前下料机构复位按钮(T)
37.00 BOOL  ; 后上料升降气缸上升按钮
37.01 BOOL  ; 后上料夹爪气缸松开按钮
37.02 BOOL  ; 后上料2级升降气缸上升按钮
37.03 BOOL  ; 后上料2级升降气缸下降按钮
37.04 BOOL  ; 后上料夹爪气缸夹紧按钮
37.05 BOOL  ; 后上料夹爪气缸松开按钮
38.00 BOOL  ; 后上料伺服归零按钮(T)
38.01 BOOL  ; 后上料伺服点动后进按钮(T)
38.02 BOOL  ; 后上料伺服点动后退按钮(T)
38.03 BOOL  ; 后上料伺服到等待位置按钮(T)
38.04 BOOL  ; 后上料伺服到取料位置按钮(T)
38.05 BOOL  ; 后上料伺服到仓3放料位置按钮(T)
38.06 BOOL  ; 后上料伺服到仓4放料位置按钮(T)
38.09 BOOL  ; 后上料伺服等待位设定按钮(T)
38.10 BOOL  ; 后上料伺服取料位设定按钮(T)
38.11 BOOL  ; 后上料伺服仓1放料位设定按钮(T)
38.12 BOOL  ; 后上料伺服仓2放料位设定按钮(T)
38.14 BOOL  ; 后上料机构单次循环按钮(T)
38.15 BOOL  ; 后上料机构复位按钮(T)
39.00 BOOL  ; 后下料升降气缸上升按钮
39.01 BOOL  ; 后下料夹爪按钮-HMI
39.02 BOOL  ; 后下料2级升降气缸上升按钮
39.03 BOOL  ; 后下料2级升降气缸下降按钮
39.04 BOOL  ; 后下料夹爪气缸夹紧按钮
39.05 BOOL  ; 后下料夹爪气缸松开按钮
39.10 BOOL  ; 腔体3检测开始位
39.11 BOOL  ; 腔体3检测结束位
39.12 BOOL  ; 腔体4检测开始位
39.13 BOOL  ; 腔体4开始位
3.00 BOOL  ; 后腔体出料伺服Ready
3.01 BOOL  ; 后腔体出料伺服Alarm
3.02 BOOL  ; 扫码阻挡气缸缩回位
3.03 BOOL  ; 扫码阻挡气缸伸出
3.04 BOOL  ; 来料隔离气缸缩回位
3.05 BOOL  ; 来料隔离气缸伸出位
3.06 BOOL  ; 上料夹爪气缸张开位
3.07 BOOL  ; 上料夹爪气缸夹紧位
3.08 BOOL  ; 进料升降伺服Ready
3.09 BOOL  ; 进料升降伺服Alarm
3.10 BOOL  ; 上料#2级升降气缸缩回位
3.11 BOOL  ; 上料#2级升降气缸伸出位
3.12 BOOL  ; 上料横移气缸伸出位
3.13 BOOL  ; 上料横移气缸缩回位
3.14 BOOL  ; 下料夹爪气缸缩回位
3.15 BOOL  ; 下料夹爪气缸伸出位
40.00 BOOL  ; 后下料伺服归零按钮(T)
40.01 BOOL  ; 后下料伺服点动后进按钮(T)
40.02 BOOL  ; 后下料伺服点动后退按钮(T)
40.03 BOOL  ; 后下料伺服到等待位置按钮(T)
40.04 BOOL  ; 后下料伺服到仓3取料位置按钮(T)
40.05 BOOL  ; 后下料伺服到仓4取料位置按钮(T)
40.06 BOOL  ; 后下料伺服到放料位置按钮(T)
40.07 BOOL  ; #1检测NG位
40.09 BOOL  ; 后下料伺服等待位设定按钮(T)
40.10 BOOL  ; 后下料伺服#3仓位设定按钮(T)
40.11 BOOL  ; 后下料伺服#4仓位设定按钮(T)
40.12 BOOL  ; 后下料伺服OK放料位设定按钮(T)
40.13 BOOL  ; 下料伺服NG放料位设定按钮(T)
40.14 BOOL  ; 后下料机构单次循环按钮(T)
40.15 BOOL  ; 后下料机构复位按钮(T)
41.00 BOOL  ; 出料#1升降气缸按钮(T)
41.01 BOOL  ; 下料3#NG放料位设定按钮
41.02 BOOL  ; 下料4#NG放料位
41.03 BOOL  ; 出料夹爪气缸张开按钮(T)
41.04 BOOL  ; #1测试N气缸按钮(T)
41.05 BOOL  ; #2测试NG气缸按钮(T)
41.06 BOOL  ; 前腔体出料顶升气缸按钮(T)
41.07 BOOL  ; 后腔体出料顶升气缸按钮(T)
41.08 BOOL  ; 出料夹爪气缸张开按钮(T)
41.09 BOOL  ; 出料夹爪气缸夹紧按钮(T)
41.10 BOOL  ; 前出料旋转气缸初位按钮(T)
41.11 BOOL  ; 前出料旋转气缸旋转按钮(T)
41.12 BOOL  ; 后出料旋转气缸初位按钮(T)
41.13 BOOL  ; 后出料旋转气缸旋转按钮(T)
41.14 BOOL  ; 前NG气缸前进按钮(T)
41.15 BOOL  ; 手动出料拉电机开关
42.00 BOOL  ; 后NG气缸前进按钮(T)
42.01 BOOL  ; 后NG气缸后退按钮(T)
42.02 BOOL  ; 下料2#NG放料位设定按钮(T)
42.03 BOOL  ; 下料3#NG放料位设定按钮(T)
42.04 BOOL  ; 下料4#NG放料位设定按钮(T)
42.10 BOOL  ; #2检测NG位
42.11 BOOL  ; #1检测NG位
42.12 BOOL  ; #2检测NG位
42.13 BOOL  ; #3检测NG位
42.14 BOOL  ; #4检测NG位
43.00 BOOL  ; 出料伺服归零按钮(T)
43.01 BOOL  ; 出料伺服点动前进按钮(T)
43.02 BOOL  ; 出料伺服点动后退按钮(T)
43.03 BOOL  ; 出料伺服到等待位置按钮(T)
43.04 BOOL  ; 出料伺服到前取料位置按钮(T)
43.05 BOOL  ; 出料伺服到后取料位置按钮(T)
43.06 BOOL  ; 出料伺服到放料位置按钮(T)
43.09 BOOL  ; 出料伺服等待位设定按钮(T)
43.10 BOOL  ; 出料伺服前取料位设定按钮(T)
43.11 BOOL  ; 出料伺服后取料位设定按钮(T)
43.12 BOOL  ; 出料伺服放料位设定按钮(T)
43.14 BOOL  ; 出料机构单次循环按钮(T)
43.15 BOOL  ; 出料机构复位按钮(T)
44.00 BOOL  ; 真空泵启动按钮(T)
44.01 BOOL  ; 真空泵停止按钮(T)
44.02 BOOL  ; 吹气启动按钮(T)
44.03 BOOL  ; 吹气停止按钮(T)
44.04 BOOL  ; 氦检仪启动按钮(T)
44.05 BOOL  ; 氦检仪停止按钮(T)
44.06 BOOL  ; #3、4真空泵启动按钮(T)
44.07 BOOL  ; 2真空泵停止按钮(T)
45.00 BOOL  ; #1腔平移气缸前进按钮(T)
45.01 BOOL  ; #1腔平移气缸后退按钮(T)
45.02 BOOL  ; #1腔顶升气缸上升按钮(T)
45.03 BOOL  ; #1腔体吹气按钮(T)
45.04 BOOL  ; #1腔密封气缸上升按钮(T)
45.05 BOOL  ; #1腔密封气缸下降按钮(T)
45.06 BOOL  ; #1腔电池抽气阀打开按钮(T)
45.07 BOOL  ; #1腔电池抽气阀关闭按钮(T)
45.08 BOOL  ; #1腔腔体抽气阀打开按钮(T)
45.09 BOOL  ; #1腔腔体抽气阀关闭按钮(T)
45.10 BOOL  ; #1腔电池破真空阀打开按钮(T)
45.11 BOOL  ; #1腔电池破真空阀关闭按钮(T)
45.12 BOOL  ; #1腔腔体破真空阀打开按钮(T)
45.13 BOOL  ; #1腔腔体破真空阀关闭按钮(T)
45.14 BOOL  ; #1腔注氦气阀打开按钮(T)
45.15 BOOL  ; #1腔注氦气阀关闭按钮(T)
46.00 BOOL  ; #1腔氦检阀打开按钮(T)
46.01 BOOL  ; #1腔氦检阀关闭按钮(T)
46.02 BOOL  ; #1腔腔体自检启动按钮(T)
46.03 BOOL  ; #1腔腔体自检停止按钮(T)
46.14 BOOL  ; #1腔机构单次循环按钮(T)
46.15 BOOL  ; #1腔机构复位按钮(T)
47.00 BOOL  ; #2腔平移气缸前进按钮(T)
47.01 BOOL  ; #2腔平移气缸后退按钮(T)
47.02 BOOL  ; #2腔顶升气缸上升按钮(T)
47.03 BOOL  ; #2腔体吹气按钮(T)
47.04 BOOL  ; #2腔密封气缸上升按钮(T)
47.05 BOOL  ; #2腔密封气缸下降按钮(T)
47.06 BOOL  ; #2腔电池抽气阀打开按钮(T)
47.07 BOOL  ; #2腔电池抽气阀关闭按钮(T)
47.08 BOOL  ; #2腔腔体抽气阀打开按钮(T)
47.09 BOOL  ; #2腔腔体抽气阀关闭按钮(T)
47.10 BOOL  ; #2腔电池破真空阀打开按钮(T)
47.11 BOOL  ; #2腔电池破真空阀关闭按钮(T)
47.12 BOOL  ; #2腔腔体破真空阀打开按钮(T)
47.13 BOOL  ; #2腔腔体破真空阀关闭按钮(T)
47.14 BOOL  ; #2腔注氦气阀打开按钮(T)
47.15 BOOL  ; #2腔注氦气阀关闭按钮(T)
48.00 BOOL  ; #2腔氦检阀打开按钮(T)
48.01 BOOL  ; #2腔氦检阀关闭按钮(T)
48.02 BOOL  ; #2腔腔体自检启动按钮(T)
48.03 BOOL  ; #2腔腔体自检停止按钮(T)
48.14 BOOL  ; #2腔机构单次循环按钮(T)
48.15 BOOL  ; #2腔机构复位按钮(T)
49.00 BOOL  ; #3腔平移气缸前进按钮(T)
49.01 BOOL  ; #3腔平移气缸后退按钮(T)
49.02 BOOL  ; #3腔顶升气缸上升按钮(T)
49.03 BOOL  ; #3腔体吹气按钮(T)
49.04 BOOL  ; #3腔密封气缸上升按钮(T)
49.05 BOOL  ; #3腔密封气缸下降按钮(T)
49.06 BOOL  ; #3腔电池抽气阀打开按钮(T)
49.07 BOOL  ; #3腔电池抽气阀关闭按钮(T)
49.08 BOOL  ; #3腔腔体抽气阀打开按钮(T)
49.09 BOOL  ; #3腔腔体抽气阀关闭按钮(T)
49.10 BOOL  ; #3腔电池破真空阀打开按钮(T)
49.11 BOOL  ; #3腔电池破真空阀关闭按钮(T)
49.12 BOOL  ; #3腔腔体破真空阀打开按钮(T)
49.13 BOOL  ; #3腔腔体破真空阀关闭按钮(T)
49.14 BOOL  ; #3腔注氦气阀打开按钮(T)
49.15 BOOL  ; #3腔注氦气阀关闭按钮(T)
4.00 BOOL  ; 出料升降伺服Ready
4.01 BOOL  ; 出料升降伺服Alarm
4.02 BOOL  ; 下料#2级升降气缸缩回位
4.03 BOOL  ; 下料#2级升降气缸伸出位
4.04 BOOL  ; 下料横移气缸伸出位
4.05 BOOL  ; 下料横移气缸缩回位
4.06 BOOL  ; 拉带进料夹爪有料感应（预留）
4.07 BOOL  ; 拉带出料夹爪有料感应（预留）
4.08 BOOL  ; 前腔体进料夹爪有料感应（预留）
4.09 BOOL  ; 前腔体出料夹爪有料感应（预留）
4.10 BOOL  ; 后腔体进料夹爪有料感应（预留）
4.11 BOOL  ; 后腔体出料夹爪有料感应（预留）
4.12 BOOL  ; 精密调压阀过低报警
4.13 BOOL  ; 后腔体出料位顶升气缸伸出位
4.14 BOOL  ; 前腔体进料夹爪张开位
4.15 BOOL  ; 前腔体进料夹爪夹紧位
50.00 BOOL  ; #3腔氦检阀打开按钮(T)
50.01 BOOL  ; #3腔氦检阀关闭按钮(T)
50.02 BOOL  ; #3腔腔体自检启动按钮(T)
50.03 BOOL  ; #3腔腔体自检停止按钮(T)
50.14 BOOL  ; #3腔机构单次循环按钮(T)
50.15 BOOL  ; #3腔机构复位按钮(T)
51.00 BOOL  ; #4腔平移气缸前进按钮(T)
51.01 BOOL  ; #4腔平移气缸后退按钮(T)
51.02 BOOL  ; #4腔顶升气缸上升按钮(T)
51.03 BOOL  ; #3腔体吹气按钮(T)
51.04 BOOL  ; #4腔密封气缸上升按钮(T)
51.05 BOOL  ; #4腔密封气缸下降按钮(T)
51.06 BOOL  ; #4腔电池抽气阀打开按钮(T)
51.07 BOOL  ; #4腔电池抽气阀关闭按钮(T)
51.08 BOOL  ; #4腔腔体抽气阀打开按钮(T)
51.09 BOOL  ; #4腔腔体抽气阀关闭按钮(T)
51.10 BOOL  ; #4腔电池破真空阀打开按钮(T)
51.11 BOOL  ; #4腔电池破真空阀关闭按钮(T)
51.12 BOOL  ; #4腔腔体破真空阀打开按钮(T)
51.13 BOOL  ; #4腔腔体破真空阀关闭按钮(T)
51.14 BOOL  ; #4腔注氦气阀打开按钮(T)
51.15 BOOL  ; #4腔注氦气阀关闭按钮(T)
52.00 BOOL  ; #4腔氦检阀打开按钮(T)
52.01 BOOL  ; #4腔氦检阀关闭按钮(T)
52.02 BOOL  ; #4腔腔体自检启动按钮(T)
52.03 BOOL  ; #4腔腔体自检停止按钮(T)
52.14 BOOL  ; #4腔机构单次循环按钮(T)
52.15 BOOL  ; #4腔机构复位按钮(T)
54.00 BOOL  ; 放料准备-拉带对接测试按钮(T)
54.01 BOOL  ; 放料完成-拉带对接测试按钮(T)
54.02 BOOL  ; 放料可移动-拉带对接测试按钮(T)
54.03 BOOL  ; 取料准备-拉带对接测试按钮(T)
54.04 BOOL  ; 取料完成-拉带对接测试按钮(T)
54.05 BOOL  ; 取料可移动-拉带对接测试按钮(T)
54.06 BOOL  ; 设备故障-拉带对接测试按钮(T)
54.10 BOOL  ; 可取料-拉带对接测试按钮(T)
54.11 BOOL  ; 可放料-拉带对接测试按钮(T)
5.00 BOOL  ; 前腔体进料升降气缸缩回位
5.01 BOOL  ; 前腔体进料升降气缸伸出位
5.02 BOOL  ; 后腔体进料夹爪张开位
5.03 BOOL  ; 后腔体进料夹爪夹紧位
5.04 BOOL  ; 后腔体进料升降气缸缩回位
5.05 BOOL  ; 后腔体进料升降气缸伸出位
5.06 BOOL  ; 前腔体出料夹爪张开位
5.07 BOOL  ; 前腔体出料夹爪夹紧位
5.08 BOOL  ; 前腔体出料升降气缸缩回位
5.09 BOOL  ; 前腔体出料升降气缸伸出位
5.10 BOOL  ; 后腔体出料夹爪张开位
5.11 BOOL  ; 后腔体出料夹爪夹紧位
5.12 BOOL  ; 后腔体出料升降气缸缩回位
5.13 BOOL  ; 后腔体出料升降气缸伸出位
5.14 BOOL  ; #1腔体移栽气缸缩回位
5.15 BOOL  ; #1腔体移栽气缸伸出位
62.00 BOOL  ; 进料升降伺归零
62.01 BOOL  ; 进料升降伺服下降点动
62.02 BOOL  ; 进料升降伺服点动上升
62.04 BOOL  ; 进料升降到取料高度
62.05 BOOL  ; 进料升降到放料高度
62.10 BOOL  ; 设为进料升降伺服取料高度
62.11 BOOL  ; 进料升降伺放料高度
6.00 BOOL  ; #1腔体顶升气缸缩回位
6.01 BOOL  ; #1腔体顶升气缸伸出位
6.02 BOOL  ; #2腔体移栽气缸缩回位
6.03 BOOL  ; #2腔体移栽气缸伸出位
6.04 BOOL  ; #2腔体顶升气缸缩回位
6.05 BOOL  ; #2腔体顶升气缸伸出位
6.06 BOOL  ; #3腔体移栽气缸缩回位
6.07 BOOL  ; #3腔体移栽气缸伸出位
6.08 BOOL  ; #3腔体顶升气缸缩回位
6.09 BOOL  ; #3腔体顶升气缸伸出位
6.10 BOOL  ; #4腔体移栽气缸缩回位
6.11 BOOL  ; #4腔体移栽气缸伸出位
6.12 BOOL  ; #4腔体顶升气缸缩回位
6.13 BOOL  ; #4腔体顶升气缸伸出位
6.14 BOOL  ; #1扫码NG推料气缸缩回位
6.15 BOOL  ; #1扫码NG推料气缸伸出位
73.00 BOOL  ; 出料升降伺服归零
73.01 BOOL  ; 出料升降伺服点动下降按钮(T)
73.02 BOOL  ; 出料升降伺服点动上升按钮
73.04 BOOL  ; 出料升降伺服到取料高度
73.05 BOOL  ; 出料升降伺服到放料高度
73.10 BOOL  ; 设出料升降取料高度
73.11 BOOL  ; 设出料升降放料高度
7.00 BOOL  ; #2扫码NG推料气缸缩回位
7.01 BOOL  ; #2扫码NG推料气缸伸出位
